	eReadMode   	: E_BACnet_CommMode;
	fCOVIncrement	: REAL;
END_STRUCT
END_TYPE

// DUTs/Types/Remote/[Internal]/ST_BACnetRM_ReqPtr
{attribute 'hide'} // [Workaround] Not hidden when lib is included

TYPE INTERNAL ST_BACnetRM_ReqPtr :
UNION
	nByte : POINTER TO BYTE;
	pPtr : PVOID;
	iReq : I_BACnetRM_BaseReq;
	
	fbBase : POINTER TO FB_BACnetRM_ReqBasic;
	fbCov : POINTER TO FB_BACnetRM_ReqCov;
	fbRead : POINTER TO FB_BACnetRM_ReqRead;
	fbRpm : POINTER TO FB_BACnetRM_ReqRpm;
	fbWrite : POINTER TO FB_BACnetRM_ReqWrite;
	fbWpm : POINTER TO FB_BACnetRM_ReqWpm;
END_UNION
END_TYPE

// DUTs/Types/Remote/[Internal]/ST_BACnetRM_RpmListEntry
{attribute 'hide'} // [Workaround] Not hidden when lib is included

{attribute 'enable_dynamic_creation'}
TYPE INTERNAL ST_BACnetRM_RpmListEntry :
STRUCT
	nEntrySize 	: DWORD;					// 0x80000000 -> next entry
	tObjectID	: T_BACnet_ObjectIdentifier;
	ePropID		: E_BACnetPropIdentifier;
	nValidBits	: DWORD;
	nArrayIndex	: DWORD;
	nPriority	: DWORD;
END_STRUCT
END_TYPE

// DUTs/Types/Remote/[Internal]/ST_BACnetRM_ScanParameter
{attribute 'hide'} // [Workaround] Not hidden when lib is included

TYPE INTERNAL ST_BACnetRM_ScanParameter :
STRUCT
	bRescrictID	 : BIT;
	bRestrictNet : BIT;
	bLocalBroadcast : BIT;
	nNetNr : UINT;
	nStartID : UDINT;
	nEndID : UDINT;
END_STRUCT
END_TYPE

// DUTs/Types/Remote/[Internal]/ST_BACnetRM_WriteEntry
{attribute 'hide'} // [Workaround] Not hidden when lib is included

{attribute 'enable_dynamic_creation'}
TYPE INTERNAL ST_BACnetRM_WriteEntry :
STRUCT
	iObject 		: I_BACnetRM_BaseObject;
	ePropID 		: E_BACnetPropIdentifier;
	
	iWriteFB 		: I_BACnetRM_BasicReq;
	
	nData 			: UDINT;
	pData 			: PVOID;
	pEnable 		: POINTER TO BOOL;
	pNull 			: POINTER TO BOOL;
	nIndex 			: UDINT := 16#FFFFFFFF;
	fCOVIncrement	: REAL := 0.0;
	nPriority 		: UDINT := 16;
END_STRUCT
END_TYPE

// DUTs/Types/Remote/ST_BACnetRM_ScanResult
TYPE ST_BACnetRM_ScanResult :
STRUCT
	tDeviceObjIdentifier	: T_BACnet_ObjectIdentifier;
	aNetAddress				: ARRAY [0..11] OF BYTE;
	nNetID					: UINT;
	{attribute 'hide'}
	nReserve1				: UINT;
	tIPAddr					: IPADDR;	
	nUDPPort				: UINT;		
	nVendorID				: UINT;
	tMaxAddr				: ETHERNET_ADDRESS;
END_STRUCT
END_TYPE

// TEST/TestPackage/Templates/HeatSupply/E_xEnergyLvl
{attribute 'qualified_only'}
TYPE E_xEnergyLvl :
(
	Protection		:= 1,
	Economy			:= 2,
	Comfort			:= 3
) UDINT;
END_TYPE

// TEST/TestPackage/Templates/HeatSupply/E_xEnergyLvlA
{attribute 'qualified_only'}
TYPE E_xEnergyLvlA :
(
	Automatic		:= 1,
	Protection		:= (E_xEnergyLvl.Protection + Automatic),
	Economy			:= (E_xEnergyLvl.Economy + Automatic),
	Comfort			:= (E_xEnergyLvl.Comfort + Automatic)
) UDINT;
END_TYPE

// GVLs/BACnet_Globals
{attribute 'qualified_only'}
VAR_GLOBAL
	{region 'Default Objects'}
		DefaultAdapter					: FB_BACnet_Adapter;									// Global linkable BACnet adapter
		DefaultServer					: FB_BACnet_Server;										// Global linkable BACnet device
	{endregion}
END_VAR
VAR_GLOBAL CONSTANT
	{region 'Commands'}
		sCmd_ConcatTitle				: STRING(5)									:= '\/';	// Command for inheriting path in entered title.
	{endregion}

	{region 'Placeholder'}
		{region 'Type Ranges'}
			nRange_ObjectTypeFirst		: INT										:= E_BACnetObjType.ObjAnalogInput;
			nRange_ObjectTypeLast		: INT										:= E_BACnetObjType.ObjChannel;
			nRange_ObjectTypeCount		: INT										:= (nRange_ObjectTypeLast - nRange_ObjectTypeFirst + 1);
		{endregion}
		{region 'Types'}
			nBACnetString_MaxLength		: INT										:= 256;
			nBACnetObjId_None			: T_BACnet_ObjectIdentifier					:= 16#FFFFFFFF;
			nBACnetInstId_Auto			: T_BACnet_ObjectIdentifier					:= 16#003FFFFF;
		{endregion}
	{endregion}

	{region 'Object specification'}
		aSpec_ObjectTypeShortcut		: ARRAY [nRange_ObjectTypeFirst .. nRange_ObjectTypeLast] OF STRING(6) := [
											(* 	AnalogInput							*)	'AI',
											(* 	AnalogOutput						*)	'AO',
											(* 	AnalogValue							*)	'AV',
											(* 	BinaryInput							*)	'BI',
											(* 	BinaryOutput						*)	'BO',
											(* 	BinaryValue							*)	'BV',
											(* 	Calendar							*)	'CAL',
											(* 	Command								*)	'CMD',
											(* 	Device								*)	'DEV',
											(* 	EventEnrollment						*)	'EE',
											(* 	File								*)	'FILE',
											(* 	Group								*)	'GROUP',
											(* 	Loop								*)	'LOOP',
											(* 	MultiStateInput						*)	'MI',
											(* 	MultiStateOutput					*)	'MO',
											(* 	NotificationClass					*)	'NC',
											(* 	Program								*)	'PROG',
											(* 	Schedule							*)	'SCHED',
											(* 	Averaging							*)	'AVG',
											(* 	MultiStateValue						*)	'MV',
											(* 	TrendLog							*)	'TLOG',
											(* 	LifeSafetyPoint						*)	'LSP',
											(* 	LifeSafetyZone						*)	'LSZ',
											(* 	Accumulator							*)	'ACC',
											(* 	PulseConverter						*)	'PC',
											(* 	EventLog							*)	'ELOG',
											(* 	GlobalGroup							*)	'GGROUP',
											(* 	TrendLogMultiple					*)	'TLM',
											(* 	LoadControl							*)	'LOAD',
											(* 	StructuredView						*)	'VIEW',
											(* 	AccessDoor							*)	'DOOR',
											(* 	<Reserved>							*)	'',
											(* 	AccessCredential					*)	'AC',
											(* 	AccessPoint							*)	'AP',
											(* 	AccessRights						*)	'AR',
											(* 	AccessUser							*)	'AU',
											(* 	AccessZone							*)	'AZ',
											(* 	CredentialDataInput					*)	'CDI',
											(* 	NetworkSecurity						*)	'NS',
											(* 	BitStringValue						*)	'BIV',
											(* 	CharacterStringValue				*)	'CV',
											(* 	DatePatternValue					*)	'DPV',
											(* 	DateValue							*)	'DV',
											(* 	DateTimePatternValue				*)	'DTPV',
											(* 	DateTimeValue						*)	'DV',
											(* 	IntegerValue						*)	'IV',
											(* 	LargeAnalogValue					*)	'LAV',
											(* 	OctetStringValue					*)	'OV',
											(* 	PositiveIntegerValue				*)	'PIV',
											(* 	TimePatternValue					*)	'TPV',
											(* 	TimeValue							*)	'TV',
											(* 	NetworkPort							*)	'NP',
											(* 	AlertEnrollment						*)	'AE',
											(* 	Channel								*)	'C'
										];
	{endregion}
	{region 'Error specification'}
		aSpec_ErrorType					: ARRAY [E_BACnet_ErrorType.First .. E_BACnet_ErrorType.Last] OF STRING := [
											(* 	eError								*)	'Error',
											(* 	eReject								*)	'Reject',
											(* 	eAbort								*)	'Abort'
										];
		aSpec_ErrorClass				: ARRAY [E_BACnet_ErrorClass.First .. E_BACnet_ErrorClass.Last] OF STRING := [
											(* 	eDevice								*)	'Device',
											(* 	eObject								*)	'Object',
											(* 	eProperty							*)	'Property',
											(* 	eResources							*)	'Resources',
											(* 	eSecurity							*)	'Security',
											(* 	eServices							*)	'Services',
											(* 	eVt									*)	'Vt',
											(* 	eCommunication						*)	'Communication'
										];
		aSpec_ErrorCode					: ARRAY [E_BACnet_ErrorCode.First .. E_BACnet_ErrorCode.Last] OF STRING := [
											(* 	eOther								*)	'Other',
											(* 	eAuthenticationFailed				*)	'Authentication failed',
											(* 	eConfigurationInProgress			*)	'Configuration in progress',
											(* 	eDeviceBusy							*)	'Device busy',
											(* 	eDynamicCreationNotSupported		*)	'Dynamic creation not supported',
											(* 	eFileAccessDenied					*)	'File access denied',
											(* 	eIncompatibleSecurityLevels			*)	'Incompatible security levels',
											(* 	eInconsistentParameters				*)	'Inconsistent parameters',
											(* 	eInconsistentSelectionCriterion		*)	'Inconsistent selection criterion',
											(* 	eInvalidDataType					*)	'Invalid data type',
											(* 	eInvalidFileAccessMethod			*)	'Invalid file access method',
											(* 	eInvalidFileStartPosition			*)	'Invalid file start position',
											(* 	eInvalidOperatorName				*)	'Invalid operator name',
											(* 	eInvalidParameterDataType			*)	'Invalid parameter data type',
											(* 	eInvalidTimeStamp					*)	'Invalid time stamp',
											(* 	eKeyGenerationError					*)	'Key generation error',
											(* 	eMissingRequiredParameter			*)	'Missing required parameter',
											(* 	eNoObjectsOfSpecifiedType			*)	'No objects of specified type',
											(* 	eNoSpaceForObject					*)	'No space for object',
											(* 	eNoSpaceToAddListElement			*)	'No space to add list element',
											(* 	eNoSpaceToWriteProperty				*)	'No space to write property',
											(* 	eNoVTSessionsAvailable				*)	'No vt sessions available',
											(* 	ePropertyIsNotAList					*)	'Property is not a list',
											(* 	eObjectDeletionNotPermitted			*)	'Object deletion not permitted',
											(* 	eObjectIdentifierAlreadyExists		*)	'ObjectIdentifier already exists',
											(* 	eOperationalProblem					*)	'Operational problem',
											(* 	ePasswordFailure					*)	'Password failure',
											(* 	eReadAccessDenied					*)	'Read access denied',
											(* 	eSecurityNotSupported				*)	'Security not supported',
											(* 	eServiceRequestDenied				*)	'Service request denied',
											(* 	eTimeout							*)	'Timeout',
											(* 	eUnknownObject						*)	'Unknown object',
											(* 	eUnknownProperty					*)	'Unknown property',
											(* 	<Reserve>							*)	'',
											(* 	eUnknownVTClass						*)	'Unknown vt class',
											(* 	eUnknownVTSession					*)	'Unknown vt session',
											(* 	eUnsupportedObjectType				*)	'Unsupported object type',
											(* 	eValueOutOfRange					*)	'Value out of range',
											(* 	eVtSessionAlreadyClosed				*)	'Vt session already closed',
											(* 	eVtSessionTerminationFailure		*)	'Vt session termination failure',
											(* 	eWriteAccessDenied					*)	'Write access denied',
											(* 	eCharacterSetNotSupported			*)	'Character set not supported',
											(* 	eInvalidArrayIndex					*)	'Invalid array index',
											(* 	eCovSubscriptionFailed				*)	'COV subscription failed',
											(* 	eNotCovProperty						*)	'Not COV property',
											(* 	eOptionalFunctionalityNotSupported	*)	'Optional functionality not supported',
											(* 	eInvalidConfigurationData			*)	'Invalid configuration data',
											(* 	eDatatypeNotSupported				*)	'Datatype not supported',
											(* 	eDuplicateName						*)	'Duplicate name',
											(* 	eDuplicateObjectId					*)	'Duplicate object ID',
											(* 	ePropertyIsNotAnArray				*)	'Property is not an array',
											(* 	eAbortBufferOverflow				*)	'Abort buffer overflow',
											(* 	eAbortInvalidAPDUInThisState		*)	'Abort invalid apdu in this state',
											(* 	eAbortPreemptedByHigherPriorityTask	*)	'Abort preempted by higher priority task',
											(* 	eAbortSegmentationNotSupported		*)	'Abort segmentation not supported',
											(* 	eAbortProprietary					*)	'Abort proprietary',
											(* 	eAbortOther							*)	'Abort other',
											(* 	eInvalidTag							*)	'Invalid tag',
											(* 	eNetworkDown						*)	'Network down',
											(* 	eRejectBufferOverflow				*)	'Reject buffer overflow',
											(* 	eRejectInconsistentParameters		*)	'Reject inconsistent parameters',
											(* 	eRejectInvalidParameterDataType		*)	'Reject invalid parameter data type',
											(* 	eRejectInvalidTag					*)	'Reject invalid tag',
											(* 	eRejectMissingRequiredParameter		*)	'Reject missing required parameter',
											(* 	eRejectParameterOutOfRange			*)	'Reject parameter out of range',
											(* 	eRejectTooManyArguments				*)	'Reject too many arguments',
											(* 	eRejectUndefinedEnumeration			*)	'Reject undefined enumeration',
											(* 	eRejectUnrecognizedService			*)	'Reject unrecognized service',
											(* 	eRejectProprietary					*)	'Reject proprietary',
											(* 	eRejectOther						*)	'Reject other',
											(* 	eUnknownDevice						*)	'Unknown device',
											(* 	eUnknownRoute						*)	'Unknown route',
											(* 	eValueNotInitialized				*)	'Value not initialized',
											(* 	eInvalidEventState					*)	'Invalid event state',
											(* 	eNoAlarmConfigured					*)	'No alarm configured',
											(* 	eLogBufferFull						*)	'Log buffer full',
											(* 	eLoggedValuePurged					*)	'Logged value purged',
											(* 	eNoPropertySpecified				*)	'No property specified',
											(* 	eNotConfiguredForTriggeredLogging	*)	'Not configured for triggered logging',
											(* 	eUnknownSubscription				*)	'Unknown subscription',
											(* 	eParameterOutOfRange				*)	'Parameter out of range',
											(* 	eListElementNotFound				*)	'List element not found',
											(* 	eBusy								*)	'Busy',
											(* 	eCommunicationDisabled				*)	'Communication disabled',
											(* 	<Reserve>							*)	38(''),
											(* 	eUnknownFileSize					*)	'Unknown file size',
											(* 	eAbortAPDUTooLong					*)	'Abort Apdu Too Long',
											(* 	eAbortApplicationExceededReplyTime	*)	'Abort Application Exceeded Reply Time',
											(* 	eAbortOutOfResources				*)	'Abort Out Of Resources',
											(* 	eAbortTsmTimeout					*)	'Abort Tsm Timeout',
											(* 	eAbortWindowSizeOutOfRange			*)	'Abort Window Size Out Of Range',
											(* 	eFileFull							*)	'File Full',
											(* 	eInconsistentConfiguration			*)	'Inconsistent Configuration',
											(* 	eInconsistentObjectType				*)	'Inconsistent object type',
											(* 	eInternalError						*)	'Internal Error',
											(* 	eNotConfigured						*)	'Not Configured',
											(* 	eOutOfMemory						*)	'Out Of Memory'
										];
		aSpec_RejectReason				: ARRAY [E_BACnet_RejectReason.First .. E_BACnet_RejectReason.Last] OF STRING := [
											(* 	eOther								*)	'Other',
											(* 	eBufferOverflow						*)	'Buffer overflow',
											(* 	eInconsistentParameters				*)	'Inconsistent parameters',
											(* 	eInvalidParameterDataType			*)	'Invalid parameter data type',
											(* 	eInvalidTag							*)	'Invalid tag',
											(* 	eMissingRequiredParameter			*)	'Missing required parameter',
											(* 	eParameterOutOfRange				*)	'Parameter out of range',
											(* 	eTooManyArguments					*)	'Too many arguments',
											(* 	eUndefinedEnumeration				*)	'Undefined enumeration',
											(* 	eUnrecognizedService				*)	'Unrecognized service'
										];
		aSpec_AbortReason				: ARRAY [E_BACnet_AbortReason.First .. E_BACnet_AbortReason.Last] OF STRING := [
											(* 	eOther								*)	'Other',
											(* 	eBufferOverflow						*)	'Buffer overflow',
											(* 	eInvalidAPDUInThisState				*)	'Invalid apdu in this state',
											(* 	ePreemptedByHigherPriorityTask		*)	'Preempted by higher priority task',
											(* 	eSegmentationNotSupported			*)	'Segmentation not supported',
											(* 	<Reserve>							*)	2(''),
											(* 	eWindowSizeOutOfRange				*)	'Window size out of range',
											(* 	eApplicationExceededReplyTime		*)	'Application exceeded reply time',
											(* 	eOutOfResources						*)	'Out of resources',
											(* 	eTSMTimeout							*)	'Tsm timeout',
											(* 	eAPDUTooLong						*)	'Apdu too long'
										];
	{endregion}
END_VAR
VAR_GLOBAL CONSTANT INTERNAL
	{region 'Placeholder'}
		{region 'AMS'}
			tInvalidAmsNetId			: T_AmsNetId						:= '0.0.0.0.0.0';
		{endregion}
		{region 'Types'}
			// (BETA) ... will be removed when ADS communication is removed
			{attribute 'hide'}
			nDataField_MaxExSchEntries			: UINT						:= 9;
			{attribute 'hide'}
			nDataField_MaxTimeValues			: UINT						:= 9;
			{attribute 'hide'}
			nDataField_MaxObjIdList				: UINT						:= 1999;
			{attribute 'hide'}
			nDataField_MaxLogBufferEntries		: UINT						:= 499;
			{attribute 'hide'}
			nDataField_MaxEventLogBufferEntries	: UINT						:= 500;
		{endregion}
	{endregion}
END_VAR

VAR_GLOBAL
	{region 'Internal'}
		// 8kByte common ADS buffer used by function blocks that access BACnet over ADS
		// [IMPORTANT] Use type "UDINT" instead of "BYTE" to ensure correct alignment!
		{attribute 'hide'}
		aDefaultBuffer					: ARRAY [0 .. (BACnet_Param.nADS_BufferSize/4)] OF UDINT;
	{endregion}
END_VAR

// GVLs/BACnet_Param
{attribute 'qualified_only'}
VAR_GLOBAL CONSTANT
	{region 'ADS'}
		tADS_TimeOut							: TIME						:= T#15S;
		nADS_BufferSize							: INT						:= 25535;								// Default 24 kByte buffer
	{endregion}
	{region 'Priorities'}
		ePrio_LifeSafety 						: E_BACnet_Priority			:= E_BACnet_Priority.eP1;
		ePrio_Critical							: E_BACnet_Priority			:= E_BACnet_Priority.eP5;
		ePrio_ManLocal							: E_BACnet_Priority			:= E_BACnet_Priority.eP7;
		ePrio_ManOperator 						: E_BACnet_Priority			:= E_BACnet_Priority.eP8;
		ePrio_Program 	 						: E_BACnet_Priority			:= E_BACnet_Priority.eP15;
		ePrio_Default	 	 					: E_BACnet_Priority			:= E_BACnet_Priority.eDefault;			// No priority used

		eRemotePrio_Default						: E_BACnet_Priority			:= E_BACnet_Priority.eP8;				// Default priority for priority enabled remote-objects
	{endregion}
		
	{region 'Event-Management'}
		sEvtMgmt_AckMsgRemote					: STRING					:= 'Acknowledged by remote user.';		// Text to indicate acknowledgement via remote access.
		sEvtMgmt_AckMsgPLC						: STRING					:= 'Acknowledged by PLC.';				// Text to indicate acknowledgement via PLC logic.
	{endregion}
	{region 'Titles'}
		sSeparator_ObjectName					: STRING					:= '_';									// Separator to be used when building Inherited object names
		sSeparator_Description					: STRING					:= ' - ';								// Separator to be used when building Inherited descriptions
		sSeparator_EventMessageText				: STRING					:= ' - ';								// Separator to be used when building Inherited event message texts
	{endregion}
		 
	{region 'Objects'}
		{region 'General'}
			nStateText_Length					: UDINT						:= 40;									// Max. count of string characters in state texts (e.g. Multustate-StateText, Binary-In/ActiveText)
			bStateText_WriteProtect				: BOOL						:= FALSE;
		{endregion}
		{region 'Multistate'}
			nMultistate_StateCount				: UDINT						:= 12;									// Count of state entries
			{attribute 'TcEncoding':='UTF-8'}
			sMultistate_DefaultStateText		: T_BACnet_StateTextArray	:= [ 'State 1', 'State 2', 'State 3' ];
		{endregion}
		{region 'Log'}  
			nLog_BufferEntryCount				: UDINT						:= 500;
					  
			nTLM_ReferenceCount					: UDINT						:= 8;
		{endregion}
		{region 'Loop'}
			nLoop_PrioForWriting				: UDINT						:= 16;
		{endregion}
		{region 'Calendar'}
			nCal_DateListCount					: INT						:= 24;									// Count of date list entries ('T_BACnet_CalendarDateList')
		{endregion}
		{region 'NC'}
			nNC_RecipientListSize				: INT						:= 8;									// Count of recipient entries
		{endregion}
		{region 'Scheduler'}
			nSched_PrioForWriting				: UDINT						:= 16;
						  
			nSched_EntryCount					: INT						:= 6;									// Count of entries in a weekday ('T_BACnet_SchedWeek') or an exception ('ST_BACnet_SchedCalendar' / 'ST_BACnet_SchedException')
			nSched_CalendarCount				: INT						:= 3;									// Count of calendar references ('T_BACnet_SchedCalendar')
			nSched_ExceptionCount				: INT						:= 24;									// Count of exceptions ('T_BACnet_SchedException')

			nSched_ReferenceCount				: UDINT						:= 2;
					  
			eSched_BType						: E_BACnet_SchedBType		:= E_BACnet_SchedBType.eBinaryPV;		// Internal datatype of boolean schedulers
		{endregion}
		{region 'Event Enrollment'}
			nEE_EventParameter_BinaryCodedSize	: UDINT						:= 100;
		{endregion}
	{endregion}
END_VAR

// TEST/TestPackage/Templates/Const
{attribute 'qualified_only'}
VAR_GLOBAL CONSTANT
	rClsZero        : REAL := 0.00001;//Comparison value to prevent a division by zero
						
	nNoActvPrio	: UDINT	:= 4294967295;//Value of the constant indicates that no priority is active	
	
	nTiSec        : UDINT := 4294966;
	nTiMin        : UDINT := 71582;

	wSUNDAY         : WORD := 0;//Constant value for Sunday
	wMONDAY         : WORD := 1;//Constant value for Monday
	wTUESDAY        : WORD := 2;//Constant value for Tuesday
	wWEDNESDAY      : WORD := 3;//Constant value for Wednesday
	wTHURSDAY       : WORD := 4;//Constant value for Thursday
	wFRIDAY         : WORD := 5;//Constant value for Friday
	wSATURDAY       : WORD := 6;//Constant value for Saturday

	TimeValue24h_ms : UDINT := 86400000;//Time value for 24 hours in ms
END_VAR

// Version/Global_Version
{attribute 'TcGenerated'}
{attribute 'no-analysis'}
{attribute 'linkalways'}
// This function has been automatically generated from the project information.
VAR_GLOBAL CONSTANT
	{attribute 'const_non_replaced'}
	stLibVersion_Tc3_BACnetRev14 : ST_LibVersion := (iMajor := 4, iMinor := 0, iBuild := 18, iRevision := 1, nFlags := 0, sVersion := '4.0.18.1');
END_VAR

// DUTs/Interfaces/Remote/Objects/[Base]/I_BACnetRM_Object
INTERFACE I_BACnetRM_Object EXTENDS I_BACnetRM_BaseObject

END_INTERFACE

// DUTs/Interfaces/Remote/Objects/[Internal]/I_BACnetRM_BaseObject
INTERFACE I_BACnetRM_BaseObject EXTENDS __SYSTEM.IQueryInterface

{attribute 'hide'}
METHOD OnCOV
VAR_INPUT
	ePropID		: E_BACnetPropIdentifier;
END_VAR
END_METHOD

{attribute 'hide'}
METHOD OnReqError
VAR_INPUT
	iRequest		: I_BACnetRM_BaseReq;
	stResult		: POINTER TO SendDataRequestResult;
	sLogCode		: STRING			:= '';
END_VAR
END_METHOD

PROPERTY Error : BOOL
GET
END_GET
END_PROPERTY

PROPERTY ObjectID : T_BACnet_ObjectIdentifier
GET
END_GET
END_PROPERTY

PROPERTY ObjectInstance : UDINT
GET
END_GET
END_PROPERTY

PROPERTY ObjectType : E_BACnetObjType
GET
END_GET
END_PROPERTY

PROPERTY ReadMode : E_BACnet_CommMode
GET
END_GET
SET
END_SET
END_PROPERTY

END_INTERFACE

// DUTs/Interfaces/Remote/Requests/[Base]/I_BACnetRM_BaseReq
{attribute 'c++_compatible'}
INTERFACE I_BACnetRM_BaseReq

{attribute 'hide'}
METHOD Send : BOOL
VAR_INPUT
END_VAR
END_METHOD

METHOD GetRequestType : E_BACnetRM_RequestType
VAR_INPUT
END_VAR
END_METHOD

METHOD IsReady : BOOL
VAR_INPUT
END_VAR
END_METHOD

END_INTERFACE

// DUTs/Interfaces/Remote/Objects/[Internal]/I_BACnetRM_ObjectOwner
{attribute 'hide'}
INTERFACE I_BACnetRM_ObjectOwner EXTENDS __SYSTEM.IQueryInterface

{attribute 'hide'}
METHOD OnBACnetRMObjectCOV
VAR_INPUT
	ePropID		: E_BACnetPropIdentifier;
END_VAR
END_METHOD

{attribute 'hide'}
METHOD OnBACnetRMObjectStateChanged
END_METHOD

{attribute 'suppress_wrn_C0410'}
{attribute 'hide'}
PROPERTY LogMsg : REFERENCE TO FB_BA_LogMessage
GET
END_GET
END_PROPERTY

END_INTERFACE

// DUTs/Interfaces/Remote/Requests/[Base]/I_BACnetRM_BasicReq
INTERFACE I_BACnetRM_BasicReq EXTENDS __SYSTEM.IQueryInterface

{attribute 'hide'}
METHOD SetError
END_METHOD

{attribute 'hide'}
METHOD SetReady
END_METHOD

END_INTERFACE

// DUTs/Interfaces/Server/[Base]/I_BACnet_Object
INTERFACE I_BACnet_Object EXTENDS I_BACnet_BaseObject

{attribute 'hide'}
PROPERTY NextSibling : I_BACnet_Object
GET
END_GET
SET
END_SET
END_PROPERTY

{attribute 'hide'}
PROPERTY PrevSibling : I_BACnet_Object
GET
END_GET
SET
END_SET
END_PROPERTY

PROPERTY IsDynamic : BOOL
GET
END_GET
END_PROPERTY

PROPERTY Parent : I_BACnet_View
GET
END_GET
SET
END_SET
END_PROPERTY

PROPERTY Description : T_MaxString
GET
END_GET
SET
END_SET
END_PROPERTY

PROPERTY ObjectName : T_MaxString
GET
END_GET
SET
END_SET
END_PROPERTY

END_INTERFACE

// DUTs/Interfaces/Server/[Internal]/I_BACnet_BaseObject
{attribute 'hide'}
INTERFACE I_BACnet_BaseObject EXTENDS I_BA_SupplementObject

{attribute 'hide'}
PROPERTY NextObject : I_BACnet_BaseObject
GET
END_GET
SET
END_SET
END_PROPERTY

PROPERTY Error : BOOL
GET
END_GET
END_PROPERTY

PROPERTY ObjectID : T_BACnet_ObjectIdentifier
GET
END_GET
END_PROPERTY

PROPERTY ObjectInstance : UDINT
GET
END_GET
END_PROPERTY

PROPERTY ObjectType : E_BACnetObjType
GET
END_GET
END_PROPERTY

PROPERTY Ready : BOOL
GET
END_GET
END_PROPERTY

METHOD ReadProperty : HRESULT
VAR_INPUT
	ePropID : E_BACnetPropIdentifier;
	pData : PVOID;
	nData : POINTER TO DINT;
END_VAR
END_METHOD

METHOD SyncPropertyCOV : BOOL
VAR_INPUT
	ePropertyID : E_BACnetPropIdentifier;
	bCOVTrig : POINTER TO BOOL;
END_VAR
END_METHOD

METHOD WriteProperty : HRESULT
VAR_INPUT
	ePropID : E_BACnetPropIdentifier;
	pData : PVOID;
	nData : DINT;
END_VAR
END_METHOD

END_INTERFACE

// DUTs/Interfaces/Server/Misc/I_BACnet_View
INTERFACE I_BACnet_View EXTENDS I_BACnet_Object

{attribute 'hide'}
METHOD AddObject : BOOL
VAR_INPUT
	iObject			: I_BACnet_Object;
END_VAR
VAR_OUTPUT
	nResultIndex	: DINT;
END_VAR
END_METHOD

{attribute 'hide'}
METHOD RemoveObject : BOOL
VAR_INPUT
	iObject			: I_BACnet_Object;
END_VAR
END_METHOD

METHOD FindObject : BOOL
VAR_INPUT
	iObject			: I_BACnet_Object;
END_VAR
VAR_IN_OUT
	nResultIndex	: DINT;
END_VAR
END_METHOD

END_INTERFACE

// DUTs/Interfaces/Server/[Internal]/I_BACnet_ObjectOwner
{attribute 'hide'}
INTERFACE I_BACnet_ObjectOwner EXTENDS __SYSTEM.IQueryInterface

{attribute 'suppress_wrn_C0410'}
{attribute 'hide'}
PROPERTY LogMsg : REFERENCE TO FB_BA_LogMessage
GET
END_GET
END_PROPERTY

{attribute 'hide'}
PROPERTY SymbolName : POINTER TO STRING
GET
END_GET
END_PROPERTY

{attribute 'hide'}
PROPERTY SymbolPath : POINTER TO T_MaxString
GET
END_GET
END_PROPERTY

{attribute 'hide'}
METHOD OnBACnetObjectStateChanged
VAR_INPUT
	tState			: TCOM_STATE;
END_VAR
END_METHOD

END_INTERFACE

// DUTs/Interfaces/Server/Misc/I_BACnet_Cal
INTERFACE I_BACnet_Cal EXTENDS I_BACnet_Object

END_INTERFACE

// POUs/Dynamic Objects/FB_BACnet_DynObjectManager
// Management of dynamically object generation.
// [Abilities]
// - Creating standard and derived objects dynamically.
// - Deleting previously created objects.
// - Automatically deletes created objects when system shuts down.
// - Automatically call created objects (Optional)
FUNCTION_BLOCK FB_BACnet_DynObjectManager
VAR_INPUT CONSTANT
	{region 'Variable Parameters'}
		{attribute 'parameterCategory':='General'}
		bCycleObjects : BOOL;								// [Optional] Call dynamically created objects cyclic (if no other calling-implementation is intended)
	{endregion}
END_VAR
VAR
	{region 'Linked Object-List'
		{attribute 'hide'}
		iFirstChild			: I_BACnet_Object;
		{attribute 'hide'}
		iLastChild			: I_BACnet_Object;
		bCreatedObjects		: UDINT;
	{endregion}
	{region 'Internal'}
		{attribute 'hide'}
		{attribute 'no_copy'}
		Server				: REFERENCE TO FB_BACnet_Server := BACnet_Globals.DefaultServer;
		{attribute 'hide'}
		nUpdateCount 		: UDINT := 0;
	{endregion}
END_VAR
VAR_STAT
	{region 'Temporary'}
		{attribute 'hide'}
		_iObj				: I_BACnet_Object;
	{endregion}	
END_VAR

// Update device:
IF (Server.nUpdateCount = nUpdateCount) THEN
	Server();
END_IF
nUpdateCount := Server.nUpdateCount;

IF (TwinCAT_SystemInfoVarList._AppInfo.ShutdownInProgress) THEN
	Reset();
ELSE
	IF (bCycleObjects) THEN
		EvaluateStructure(E_BACnet_EvaluationMode.eCycle, 0, TRUE);
	END_IF
END_IF

METHOD PRIVATE EvaluateStructure
VAR_INPUT
	eMode			: E_BACnet_EvaluationMode;
	iObject			: I_BACnet_Object			:= 0;
	bRecursive		: BOOL						:= FALSE;
END_VAR
VAR
	_iObj			: I_BACnet_Object;
	_iTemp			: I_BACnet_Object;
	_fbView			: POINTER TO FB_BACnet_View;
END_VAR
VAR_STAT
	{region 'Temporary'}
		{attribute 'hide'}
		_fbObject	: POINTER TO FB_BACnet_Object;
	{endregion}	
END_VAR
IF (iObject = 0) THEN
	// Iterate though root objects:
	_iObj := iFirstChild;
	WHILE (_iObj <> 0) DO
		_iTemp := _iObj.NextSibling;
		THIS^.EvaluateStructure(eMode, _iObj, bRecursive);
		_iObj := _iTemp;
	END_WHILE;
ELSE
	// Pre-Evaluation treatment:
	CASE (eMode) OF
		E_BACnet_EvaluationMode.eCycle:
			iObject.OnCycle(FALSE);
	END_CASE
	
	IF (bRecursive) AND_THEN (iObject.ObjectType = E_BACnetObjType.ObjStructuredView) AND_THEN (__QUERYPOINTER(iObject, _fbView)) THEN
		// Iterate though child-objects of 'iObject':
		_iObj := _fbView^.iFirstChild;
		WHILE (_iObj <> 0) DO
			_iTemp := _iObj.NextSibling;
			THIS^.EvaluateStructure(eMode, _iObj, bRecursive);
			_iObj := _iTemp;
		END_WHILE;
	END_IF
	
	// Post-Evaluation treatment:
	CASE (eMode) OF
		E_BACnet_EvaluationMode.eDeleteObjects:
			IF (__QUERYPOINTER(iObject, _fbObject)) THEN
				DeleteObjectEx(_fbObject);
			END_IF
	END_CASE
END_IF
END_METHOD

METHOD PRIVATE DeleteObjectEx
VAR_INPUT
	fbObject			: POINTER TO FB_BACnet_Object;
END_VAR
VAR
	_iSrv				: POINTER TO ITcIoBACnetPlcServer;
	_iObj				: POINTER TO ITcIoBACnetPlcObject;
END_VAR
_iSrv := ADR(fbObject^.ipSrv);
_iObj := ADR(fbObject^.ipObj);

IF (_iSrv^.DeletePlcObjectRT(_iObj) <> S_OK) THEN
	F_BA_LogMessage1(ADSLOG_MSGTYPE_WARN, 'DO46', 'Dynamic PLC object deleted, but failed to delete object "%s" from stack!', F_STRING(fbObject^.sObjectName));
END_IF

__DELETE(fbObject);
bCreatedObjects := (bCreatedObjects-1);
END_METHOD

// Called after online change.
{attribute 'call_after_online_change_slot' := '10'}
METHOD PROTECTED OnPostOnlineChange
Reset();
END_METHOD

// Create an object dynamically.
METHOD CreateObject : BOOL
VAR_IN_OUT
	fbResult			: POINTER TO FB_BACnet_Object;
END_VAR
VAR_INPUT
	eObjectType			: E_BACnet_CreateObjType;
	nObjectInstance		: UDINT							:= BACnet_Globals.nBACnetInstId_Auto;
	sObjectName			: T_MaxString;
	sDescription		: T_MaxString;
	fbParent			: POINTER TO FB_BACnet_View		:= 0;
END_VAR
VAR
	_uObj				: U_BACnet_CreateObj;
END_VAR
// Evaluate type:
CASE (eObjectType) OF
	E_BACnet_CreateObjType.eAnalogInputRaw:			_uObj.AIRaw := __NEW(FB_BACnet_AI_Raw);
	E_BACnet_CreateObjType.eAnalogOutputRaw:		_uObj.AORaw := __NEW(FB_BACnet_AO_Raw);
	E_BACnet_CreateObjType.eAnalogOutputRaw5P:		_uObj.AORaw5P := __NEW(FB_BACnet_AO_Raw5P);
	E_BACnet_CreateObjType.eAnalogValue:			_uObj.AV := __NEW(FB_BACnet_AV);
	E_BACnet_CreateObjType.eAnalogValue5P:			_uObj.AV5P := __NEW(FB_BACnet_AV_5P);
	E_BACnet_CreateObjType.eAnalogValueDisp:		_uObj.AVDisp := __NEW(FB_BACnet_AV_Disp);
	E_BACnet_CreateObjType.eAnalogValueSetp:		_uObj.AVSetp := __NEW(FB_BACnet_AV_Setp);
	
	E_BACnet_CreateObjType.eBinaryInputRaw:			_uObj.BIRaw := __NEW(FB_BACnet_BI_Raw);
	E_BACnet_CreateObjType.eBinaryOutputRaw:		_uObj.BORaw := __NEW(FB_BACnet_BO_Raw);
	E_BACnet_CreateObjType.eBinaryOutputRaw5P:		_uObj.BORaw5P := __NEW(FB_BACnet_BO_Raw5P);
	E_BACnet_CreateObjType.eBinaryValue:			_uObj.BV := __NEW(FB_BACnet_BV);
	E_BACnet_CreateObjType.eBinaryValue5P:			_uObj.BV5P := __NEW(FB_BACnet_BV_5P);
	E_BACnet_CreateObjType.eBinaryValueDisp:		_uObj.BVDisp := __NEW(FB_BACnet_BV_Disp);
	E_BACnet_CreateObjType.eBinaryValueSetp:		_uObj.BVSetp := __NEW(FB_BACnet_BV_Setp);
	
	E_BACnet_CreateObjType.eMultistateInputRaw:		_uObj.MIRaw := __NEW(FB_BACnet_MI_Raw);
	E_BACnet_CreateObjType.eMultistateOutputRaw:	_uObj.MORaw := __NEW(FB_BACnet_MO_Raw);
	E_BACnet_CreateObjType.eMultistateOutputRaw5P:	_uObj.MORaw5P := __NEW(FB_BACnet_MO_Raw5P);
	E_BACnet_CreateObjType.eMultistateValue:		_uObj.MV := __NEW(FB_BACnet_MV);
	E_BACnet_CreateObjType.eMultistateValue5P:		_uObj.MV5P := __NEW(FB_BACnet_MV_5P);
	E_BACnet_CreateObjType.eMultistateValueDisp:	_uObj.MVDisp := __NEW(FB_BACnet_MV_Disp);
	E_BACnet_CreateObjType.eMultistateValueSetp:	_uObj.MVSetp := __NEW(FB_BACnet_MV_Setp);
	
	E_BACnet_CreateObjType.eCalendar:				_uObj.Clnd := __NEW(FB_BACnet_Cal);
	E_BACnet_CreateObjType.eDevice:					_uObj.Device := __NEW(FB_BACnet_Device);
	E_BACnet_CreateObjType.eFile:					_uObj.File := __NEW(FB_BACnet_File);
	E_BACnet_CreateObjType.eLoop:					_uObj.Loop := __NEW(FB_BACnet_Loop);
	E_BACnet_CreateObjType.eNotificationClass:		_uObj.NC := __NEW(FB_BACnet_NC);
	E_BACnet_CreateObjType.eProg:					_uObj.Prog := __NEW(FB_BACnet_Prog);
	E_BACnet_CreateObjType.eScheduleAnalog:			_uObj.SchedA := __NEW(FB_BACnet_SchedA);
	E_BACnet_CreateObjType.eScheduleBinary:			_uObj.SchedB := __NEW(FB_BACnet_SchedB);
	E_BACnet_CreateObjType.eScheduleMultistate:		_uObj.SchedM := __NEW(FB_BACnet_SchedM);
	E_BACnet_CreateObjType.eAccumulator:			_uObj.Acc := __NEW(FB_BACnet_Acc);
	E_BACnet_CreateObjType.ePulseConverter:			_uObj.PC := __NEW(FB_BACnet_PC);
	E_BACnet_CreateObjType.eStructuredView:			_uObj.View := __NEW(FB_BACnet_View);

ELSE
	F_BA_LogMessage1(ADSLOG_MSGTYPE_ERROR, 'CO20', 'Unsupported object type "%d"!', F_INT(eObjectType));
	RETURN;
END_CASE

IF (_uObj.Obj = 0) THEN
	F_BA_LogMessage1(ADSLOG_MSGTYPE_ERROR, 'CO25', 'Unknown error on creating dynamic object of type "%d"!', F_INT(eObjectType));
ELSE
	IF (CreateObjectEx(_uObj.Obj, nObjectInstance, sObjectName, sDescription, fbParent)) THEN
		fbResult := _uObj.Obj;
		CreateObject := TRUE;
	ELSE
		__DELETE (_uObj.Obj);
		fbResult := 0;
	END_IF
END_IF
END_METHOD

// Create an object dynamically.
// > 'fbResult' is an object, that was previously created with '__NEW()'.
//   Useful if 'fbResult' is a derived object type.
METHOD CreateObjectEx : BOOL
VAR_INPUT
	fbObject			: POINTER TO FB_BACnet_Object;
	nObjectInstance		: UDINT							:= BACnet_Globals.nBACnetInstId_Auto;
	sObjectName			: T_MaxString;
	sDescription		: T_MaxString;
	fbParent			: POINTER TO FB_BACnet_View		:= 0;
END_VAR
IF (Ready) THEN
	IF (fbObject = 0) THEN
		F_BA_LogMessage(ADSLOG_MSGTYPE_ERROR, 'CO02', 'Invalid object!');
	ELSIF (sObjectName = '') THEN
		F_BA_LogMessage1(ADSLOG_MSGTYPE_ERROR, 'CO04', 'Unable to create object due to invalid name "%s"!', F_STRINGEx(sObjectName));
	ELSIF (sDescription = '') THEN
		F_BA_LogMessage1(ADSLOG_MSGTYPE_ERROR, 'CO06', 'Unable to create object due to invalid description "%s"!', F_STRINGEx(sDescription));
	ELSIF (fbParent <> 0) AND_THEN (NOT fbParent^.IsDynamic) THEN
		F_BA_LogMessage1(ADSLOG_MSGTYPE_ERROR, 'CO08', 'Refused to create object of non-dynamic parent "%s"!', F_STRING(fbParent^.SymbolPath^));
	ELSE
		IF (fbObject^.DynamicInit(THIS, nObjectInstance, sObjectName, sDescription, fbParent)) THEN
			IF (fbParent = 0) THEN
				// Append linked object list:
				IF (iFirstChild = 0) THEN
					iFirstChild := fbObject^;
				ELSE
					iLastChild.NextSibling := fbObject^;
				END_IF
				iLastChild := fbObject^;
			END_IF
		
			bCreatedObjects := (bCreatedObjects+1);
			CreateObjectEx := TRUE;
		END_IF
	END_IF
END_IF
END_METHOD

// Delete a dynamically created object.
// > IMPORTANT: Pointers to deleted objects are invalid!
METHOD DeleteObject : BOOL
VAR_IN_OUT
	fbObject			: POINTER TO FB_BACnet_Object;
END_VAR
VAR
	_fbView				: POINTER TO FB_BACnet_View;
	_fbObject			: POINTER TO FB_BACnet_Object;
	_iObject			: I_BACnet_Object;
END_VAR
IF (fbObject = 0) THEN
	F_BA_LogMessage(ADSLOG_MSGTYPE_ERROR, 'DO02', 'Invalid dynamic object!');
ELSIF (NOT fbObject^.IsDynamic) THEN
	F_BA_LogMessage1(ADSLOG_MSGTYPE_ERROR, 'DO04', 'Refused to delete non-dynamic object "%s"!', F_STRING(fbObject^.SymbolPath^));
ELSIF (fbObject^.fbDynProducer <> THIS) THEN
	F_BA_LogMessage1(ADSLOG_MSGTYPE_ERROR, 'DO06', 'Refused to delete dynamic object "%s" that is not created by current object manager!', F_STRING(fbObject^.SymbolPath^));
ELSE
	IF (fbObject^.ObjectType = E_BACnetObjType.ObjStructuredView) THEN
		_fbView := fbObject;
		IF (_fbView^.iFirstChild <> 0) THEN
			F_BA_LogMessage1(ADSLOG_MSGTYPE_ERROR, 'DO11', 'Unable to delete dynamic object "%s" because it has existing child objects!', F_STRING(fbObject^.SymbolPath^));
			RETURN;
		END_IF
	END_IF
	
	_fbObject := fbObject;
	_iObject := _fbObject^;
	
	IF (_fbObject^.iParent = 0) THEN
		// Remove object from linked object list of current instance:
		fbObject^.RemoveFromLinkedObjList(iFirstChild, iLastChild);
	ELSE
		// Remove object from parent:
		_fbObject^.iParent.RemoveObject(_iObject);
	END_IF
	
	DeleteObjectEx(_fbObject);
	fbObject := 0;
	
	DeleteObject := TRUE;
END_IF
END_METHOD

PROPERTY Ready : BOOL
GET
Ready := Server.Operational;
END_GET
END_PROPERTY

// Delete all dynamically created objects.
METHOD Reset
// Delete all created objects:
EvaluateStructure(E_BACnet_EvaluationMode.eDeleteObjects, 0, TRUE);

iFirstChild := 0;
iLastChild := 0;
bCreatedObjects := 0;
END_METHOD

PROPERTY CreatedObjects : UDINT
GET
CreatedObjects := bCreatedObjects;
END_GET
END_PROPERTY

METHOD FB_exit : BOOL
VAR_INPUT
	bInCopyCode : BOOL; // if TRUE, the exit method is called for exiting an instance that is copied afterwards (online change).
END_VAR
Reset();
END_METHOD

END_FUNCTION_BLOCK

// POUs/Local/FB_BACnet_Server
{attribute 'no_assign'}
FUNCTION_BLOCK FB_BACnet_Server
VAR_INPUT
	bWritePersistent		: BOOL;
END_VAR
VAR_INPUT CONSTANT
	{region 'Fixed Parameters'}
		{attribute 'parameterCategory':='General'}
		Adapter	: REFERENCE TO FB_BACnet_Adapter := BACnet_Globals.DefaultAdapter;
	{endregion}
END_VAR
VAR_INPUT CONSTANT PERSISTENT
	{region 'Variable Parameters'}
		{attribute 'parameterCategory':='General'}
		bSupportBackup : BOOL;							// Support backup of PLC persistent data when BACnet backup service is used
		{attribute 'parameterCategory':='General'}
		bDisableWOC : BOOL;								// Deactivate write-on-change mechanism
		{attribute 'parameterCategory':='General'}
		tAmsPort : T_AmsPort := 1000;					// Default port when port can not be determined automatically
	{endregion}
END_VAR
VAR_INPUT CONSTANT
	{region 'Operational Parameters'}
		{attribute 'parameterCategory':='General'}
		bReset : BOOL;									// Manual trigger to reset errors
		{attribute 'parameterCategory':='General'}
		tWritePersistent : TIME := T#30M;				// Cyclic write persistent data
	{endregion}
END_VAR
VAR_OUTPUT
	nRev					: DINT := -1;				// Protocol revision no.
	stAdsConn				: ST_BACnet_AdsConnection;
	eSysStatus				: E_BACnet_DeviceStatus;
	eState					: E_BACnet_ServerState	:= E_BACnet_ServerState.eInitServer;
	bBackupAct				: BOOL;
	bWritePersisAct			: BOOL;
	bWOCDisabled			: BOOL;
	eErrorID				: E_BACnet_Error;
END_VAR
VAR
	{region 'General'}
		nUpdateCount	 	: UDINT := 0;
	{endregion}
	{region 'Object List'}
		{attribute 'hide'}
		ipFirstObject		: I_BACnet_BaseObject;
		{attribute 'hide'}
		ipLastObject		: I_BACnet_BaseObject;
		{attribute 'hide'}
		nObjectCount		: UDINT;
	{endregion}
	{region 'Interface Pointer'}
		{attribute 'hide'}
		oServerOID			: OTCID; 
		{attribute 'hide'}
		iServer 			: ITcIoBACnetPlcServer;
		{attribute 'hide'}
		iDevice				: ITcIoBACnetPlcDevice;
		{attribute 'hide'}
		oDeviceOID			: OTCID;
		{attribute 'hide'}
		iObject				: ITcIoBACnetPlcObject;
	{endregion}
	{region 'Internal'}
		_ObjectId			: DWORD;	
		_ServerStatus		: WORD;
		_ServerControl		: WORD;
		_fbWritePersistent	: FB_WritePersistentData	:= (PORT:=TwinCAT_SystemInfoVarList._AppInfo.AdsPort, TMOUT:=T#1S, MODE:=E_PersistentMode.SPDM_2PASS);
		_rtrigBackup		: R_TRIG;
		_rtrigReset			: R_TRIG;
		_rtrigWritePers		: R_TRIG;
		_ePersDataState		: E_BACnet_PersistentDataState;
		_nPlcPort			: T_AmsPort;
		_tCyclicWrPers		: TON;
	{endregion}
	{region 'Misc'}
		{attribute 'hide'}
		fbLogMsg			: FB_BA_LogMessage;
	{endregion}
	{region 'Temporary'}
		_hResult			: HRESULT;
	{endregion}
END_VAR

IF (__ISVALIDREF(Adapter)) THEN
	Adapter();
END_IF
// Remind current number of update counter:
nUpdateCount := Adapter._nUpdateCount;

CASE (eState) OF
	E_BACnet_ServerState.eInitServer:
		eErrorID := E_BACnet_Error.eNoError;
		
		// Check if NetID is plausible:
		IF (Adapter.sAmsNetId = '') THEN
			fbLogMsg.Show1(ADSLOG_MSGTYPE_ERROR, 'D20', 'Configured AMS-NetID "%s" is invalid!', F_STRINGEx(Adapter.sAmsNetId), FALSE);
			eErrorID := E_BACnet_Error.eNoValidNetId;
		ELSIF (Adapter.eDevState <= E_BACnet_AdapterStatus.eInit) THEN
			; // Wait for adapter to get initialized.
		ELSIF (iDevice = 0) THEN
			Reset();
			iDevice := Adapter.Device;
			IF (iDevice <> 0) THEN
				iDevice.TcAddRef();
				iDevice.GetDeviceData(ADR(TwinCAT_SystemInfoVarList._AppInfo.ObjId), SIZEOF(OTCID), E_BACnet_DeviceData.eSetPlcOID);
			END_IF
		END_IF
		
		IF (iServer = 0) THEN
			IF (iDevice <> 0) THEN
				_hResult := iDevice.GetClientById(16#FFFFFFFF, ADR(iServer));
			ELSIF (oServerOID <> 0) THEN
				_hResult := FW_ObjMgr_GetObjectInstance(oid:=oServerOID, iid:=TC_GLOBAL_IID_LIST.IID_ITcIoBACnetPlcServer, pipUnk:=ADR(iServer));
			ELSE
				_hResult := S_OK;
			END_IF
			IF (iServer <> 0) THEN
				_hResult := iServer.GetAdsPort(ADR(tAmsPort));
				
				// Get Device-Object:
				IF (SUCCEEDED(_hResult)) THEN
					_hResult := iServer.GetObjectByObjectId(ADR(iObject), 16#23FFFFF);
					IF (SUCCEEDED(_hResult)) THEN
						_hResult := SEL(ReadPropertyUDInt(E_BACnetPropIdentifier.PropObjectIdentifier, _ObjectId), E_FAIL, S_OK);
					END_IF
					IF (SUCCEEDED(_hResult)) THEN
						_hResult := iObject.GetPropertyValue(E_BACnetPropIdentifier.PropProtocolRevision, ADR(nRev), 0);
					END_IF
					eErrorID := SEL(SUCCEEDED(_hResult), E_BACnet_Error.eInvalidServer, E_BACnet_Error.eNoError);
				END_IF
				
				// Indicate stack begin of object initialization: 
				_hResult := iServer.OnPlcAction(E_BACnet_PlcAction.eStart);
				IF (SUCCEEDED(_hResult)) THEN
					oDeviceOID := iServer.GetBACnetDeviceOid();
					IF (oDeviceOID = 0) THEN
						fbLogMsg.Show(ADSLOG_MSGTYPE_ERROR, 'D47', 'Internal error!', FALSE);
						eErrorID:=E_BACnet_Error.eInvalidServer;
					ELSE
						FW_ObjMgr_GetObjectInstance(oid:=oDeviceOID, iid:=TC_GLOBAL_IID_LIST.IID_ITcIoBACnetPlcDevice, pipUnk:=ADR(iDevice));
						
						// Start initializing objects:
						eState := E_BACnet_ServerState.eInitDefObjs;
					END_IF
				ELSE
					IF (iDevice = 0) THEN
						eErrorID := E_BACnet_Error.eInvalidTask;
						fbLogMsg.Show(ADSLOG_MSGTYPE_ERROR, 'D56', 'Task configuration invalid!', FALSE);
					ELSE
						fbLogMsg.Show1(ADSLOG_MSGTYPE_ERROR, 'D60', 'Internal error "0x%x"!', F_DINT(_hResult), FALSE);
						eErrorID := E_BACnet_Error.eInvalidServer;
					END_IF
					FW_SafeRelease(ADR(iServer));
					iServer:=0;				
				END_IF
			ELSE
				IF (_hResult = S_OK) THEN
					; // Resolving server...
				ELSE
					eErrorID := E_BACnet_Error.eInvalidServer;
					CASE (F_BACnet_FilterErrCode(_hResult)) OF
						E_AdsErr.DEVICE_NOTFOUND:
							fbLogMsg.Show(ADSLOG_MSGTYPE_ERROR, 'D74', 'BACnet-Server configuration missing!', FALSE);
					ELSE
						fbLogMsg.Show1(ADSLOG_MSGTYPE_ERROR, 'D78', 'BACnet-Server configuration invalid (Result: "0x%x")!', F_DINT(_hResult), FALSE);
					END_CASE
				END_IF
			END_IF
		END_IF
		
	E_BACnet_ServerState.eInitDefObjs:
		// [Hint] Initialization of defined objects DONE at this step.
		eState := E_BACnet_ServerState.eInitUndefObjs;
	
	E_BACnet_ServerState.eInitUndefObjs:
		// [Hint] Initialization of undefined objects DONE at this step.
		eState := E_BACnet_ServerState.eInitDefRefObjs;
	
	E_BACnet_ServerState.eInitDefRefObjs:
		// [Hint] Initialization of referring, defined objects DONE at this step.
		eState := E_BACnet_ServerState.eInitUndefRefObjs;
	
	E_BACnet_ServerState.eInitUndefRefObjs:
		// [Hint] Initialization of referring, undefined objects DONE at this step.
		
		_hResult := iServer.OnPlcAction(E_BACnet_PlcAction.eCreateFinish);
		IF (NOT SUCCEEDED(_hResult)) THEN
			fbLogMsg.Show1(ADSLOG_MSGTYPE_ERROR, 'D82', 'Internal error "0x%x"!', F_DINT(_hResult), FALSE);
			eErrorID := E_BACnet_Error.eInvalidServer;
		ELSIF (NOT Valid) THEN
			fbLogMsg.Show(ADSLOG_MSGTYPE_ERROR, 'D85', 'Invalid Server parameters!', FALSE);
			eErrorID := E_BACnet_Error.eInvalidParameter;
		ELSE
			// Validate user settings:
			IF (NOT F_BACnet_IsSchedBTypeValid(BACnet_Param.eSched_BType)) THEN
				fbLogMsg.Show(ADSLOG_MSGTYPE_ERROR, 'S90', 'Global parameter "eSchedB_Type" is invalid!', FALSE);
			END_IF
	
			eState := E_BACnet_ServerState.eOperation;
		END_IF
	
	E_BACnet_ServerState.eOperation:
		// Read properties:
		ReadPropertyInt(E_BACnetPropIdentifier.PropSystemStatus, eSysStatus);
		ReadPropertyInt(E_BACnetPropIdentifier.PropPersistentData, _ePersDataState);
		
		// Refresh server state:
		iServer.UpdateDeviceStatus(ADR(_ServerControl), ADR(_ServerStatus));
		bWOCDisabled := ((_ServerStatus AND 16#0004) = 16#0004);

		// Backup (Trigger writing of persistent data):
		_rtrigWritePers(CLK := bWritePersistent);
		_tCyclicWrPers(IN := (NOT _fbWritePersistent.BUSY), PT := tWritePersistent);
		
		IF (_fbWritePersistent.START) THEN
			IF (NOT _fbWritePersistent.BUSY) THEN
				// Writing persistent data finished:
				_ServerControl.1 := TRUE;
				_fbWritePersistent.START := FALSE;
			END_IF
		ELSE
			_ServerControl.1 := FALSE;
			_fbWritePersistent.START :=
				(eSysStatus = E_BACnet_DeviceStatus.eBackupInProgress) OR_ELSE
				(_ePersDataState = E_BACnet_PersistentDataState.eWrite) OR_ELSE
				(_rtrigWritePers.Q) OR_ELSE
				(_tCyclicWrPers.Q);
		END_IF
		_fbWritePersistent(BUSY=>bBackupAct);
		
	E_BACnet_ServerState.Invalid:
		;
		
ELSE
	fbLogMsg.Show1(ADSLOG_MSGTYPE_ERROR, 'S100', 'Invalid server state "%d"!', F_BYTE(eState), FALSE);
	eErrorID := E_BACnet_Error.eInvalidParameter;
END_CASE

IF (Error) THEN
	IF (eState = E_BACnet_ServerState.Invalid) THEN
		// Error occured in past cycles.
		
		// Reset Trigger:
		_rtrigReset(CLK:=bReset);
		IF (_rtrigReset.Q) OR_ELSE ((eErrorID < E_BACnet_Error.FirstResetError) OR (eErrorID >= E_BACnet_Error.LastResetError)) THEN
			_rtrigReset(CLK:=FALSE);
			Reset();
		END_IF
	ELSE
		// Error occured this cycle.
		Reset();
		eState := E_BACnet_ServerState.Invalid;
	END_IF
END_IF

// Control:
_ServerControl.2 := bDisableWOC;		// Disable write-on-change
_ServerControl.11 := Operational;		// PLC running - process data valid

{attribute 'hide'}
METHOD GetObjectByID : BOOL
VAR_INPUT
	tObjectID	: T_BACnet_ObjectIdentifier;
END_VAR
VAR_OUTPUT
	iResult		: I_BACnet_BaseObject;
END_VAR
iResult := ipFirstObject;
WHILE (iResult <> 0) DO
	IF (iResult.ObjectID = tObjectID) THEN
		GetObjectByID := TRUE;
		RETURN;
	END_IF
	iResult := iResult.NextObject;
END_WHILE
END_METHOD

{attribute 'hide'}
METHOD RegisterObject : BOOL
VAR_INPUT
	iObject	  : I_BACnet_BaseObject;
END_VAR
IF (iObject <> 0) THEN
	IF (nObjectCount = 0) THEN
		ipFirstObject := iObject;
	ELSE
		ipLastObject.NextObject := iObject;
	END_IF
	ipLastObject := iObject;
	nObjectCount := (nObjectCount + 1);
	
	RegisterObject := TRUE;
END_IF
END_METHOD

{attribute 'hide'}
PROPERTY ObjectCount : UDINT
GET
VAR
	cnt : UDINT;
END_VAR
IF iObject = 0 THEN
	ObjectCount:=0;
	RETURN;
END_IF

IF S_OK = iObject.SyncReadProperty(E_BACnetPropIdentifier.PropObjectList, ADR(cnt), 0, 0) THEN
 	ObjectCount:=cnt;
	RETURN;
END_IF

ObjectCount:=0;
END_GET
END_PROPERTY

{attribute 'hide'}
PROPERTY ServerItf : ITcIoBACnetPlcServer
GET
ServerItf := iServer;
END_GET
END_PROPERTY

METHOD PRIVATE Reset
IF iServer <> 0 THEN
	iServer.OnPlcAction(E_BACnet_PlcAction.eSuspend); // SUSPEND - delete all pointers to PLC
	FW_SafeRelease(ADR(iServer));
	iServer:=0;
END_IF
IF iObject <> 0 THEN
	FW_SafeRelease(ADR(iObject));
	iObject:=0;
END_IF	
IF iDevice <> 0 THEN
	FW_SafeRelease(ADR(iDevice));
	iDevice:=0;
END_IF 

// Object List:
ipLastObject := 0;
nObjectCount := 0;

eState := E_BACnet_ServerState.eInitServer;
eSysStatus := E_BACnet_DeviceStatus.Invalid;
bWOCDisabled := FALSE;
END_METHOD

// Called after online change.
{attribute 'call_after_online_change_slot' := '10'}
METHOD PROTECTED OnPostOnlineChange
Reset();
END_METHOD

PROPERTY Error : BOOL
GET
Error := (eErrorID <> E_BACnet_Error.eNoError);
END_GET
END_PROPERTY

PROPERTY Operational : BOOL
GET
Operational := (eState=E_BACnet_ServerState.eOperation);
END_GET
END_PROPERTY

PROPERTY Valid : BOOL
GET
Valid := (_ObjectId <> 16#00000000);
END_GET
END_PROPERTY

{attribute 'hide'}
METHOD ReadPropertyInt : BOOL
VAR_INPUT
	ePropID : E_BACnetPropIdentifier;
	value : REFERENCE TO INT;
END_VAR
VAR_STAT
	_hr : HRESULT;
	_val : DINT;
	_size : DINT := SIZEOF(_val);
END_VAR
IF iObject<>0 AND (__ISVALIDREF(value)) THEN
	_hr:=iObject.SyncReadProperty(TO_INT(ePropID), ADR(_val), ADR(_size), 16#FFFFFFFF);
	IF (_hr = S_OK) THEN
		value := TO_INT(_val);
		ReadPropertyInt:=TRUE;
		RETURN;
	END_IF
END_IF
ReadPropertyInt:=FALSE;
END_METHOD

{attribute 'hide'}
METHOD ReadPropertyUDInt : BOOL
VAR_INPUT
	ePropID : E_BACnetPropIdentifier;
	value : REFERENCE TO UDINT;
END_VAR
VAR
	_hr : HRESULT;
	_size : DINT := 4;
END_VAR
IF iObject<>0 AND (__ISVALIDREF(value)) THEN
	_hr:=iObject.SyncReadProperty(TO_INT(ePropID), ADR(value), ADR(_size), 16#FFFFFFFF);
	IF (_hr = S_OK) THEN
		ReadPropertyUDInt:=TRUE;
		RETURN;
	END_IF
END_IF
ReadPropertyUDInt:=FALSE;
END_METHOD

METHOD FB_Exit : BOOL
VAR_INPUT
	 bInCopyCode : BOOL; // if TRUE, the exit method is called for exiting an instance that is copied afterwards (online change).
END_VAR
Reset();
END_METHOD

END_FUNCTION_BLOCK

// POUs/Helper/[internal]/F_BACnet_FilterErrCode
{attribute 'hide'}
FUNCTION F_BACnet_FilterErrCode : HRESULT
VAR_INPUT
	hResult		: HRESULT;
END_VAR

F_BACnet_FilterErrCode := TO_UINT(hResult) AND 16#FFF;

END_FUNCTION

// POUs/Helper/[internal]/Validation-Functions/F_BACnet_IsSchedBTypeValid
{attribute 'hide'}
FUNCTION F_BACnet_IsSchedBTypeValid : BOOL
VAR_INPUT
	eType		: E_BACnet_SchedBType;
END_VAR

F_BACnet_IsSchedBTypeValid := ((E_BACnet_SchedBType.First <= eType) AND_THEN (eType <= E_BACnet_SchedBType.Last));

END_FUNCTION

// TEST/TestPackage/BACKUP
PROGRAM BACKUP
VAR
	cfgTsZip	: FB_BACnet_File := (bEnBackupFile:=TRUE, sObjectName := 'CurrentConfig.tszip',	sFileName := 'CurrentConfig.tszip');
	plcBootdata : FB_BACnet_File := (bEnBackupFile:=TRUE, sObjectName := 'Port_851.bootdata', 	sFileName := 'Plc\Port_851.bootdata');
	plcApp 		: FB_BACnet_File := (bEnBackupFile:=TRUE, sObjectName := 'Port_851.app', 		sFileName := 'Plc\Port_851.app');
	plcCrc 		: FB_BACnet_File := (bEnBackupFile:=TRUE, sObjectName := 'Port_851.crc', 		sFileName := 'Plc\Port_851.crc');
	plcTiZip	: FB_BACnet_File := (bEnBackupFile:=TRUE, sObjectName := 'Port_851_boot.tizip', sFileName := 'Plc\Port_851_boot.tizip');
END_VAR

cfgTsZip();
plcBootdata();
plcApp();
plcCrc();
plcTiZip();

END_PROGRAM

// POUs/Local/Objects/FB_BACnet_File
// File Object
{attribute 'enable_dynamic_creation'}
FUNCTION_BLOCK FB_BACnet_File EXTENDS FB_BACnet_Object
VAR_INPUT CONSTANT 
	{region 'Fixed Parameters'}
		{attribute 'parameterCategory':='General'}
		bEnBackupFile : BOOL;
		{attribute 'parameterCategory':='General'}
		{attribute 'TcEncoding':='UTF-8'}
		sFileName : T_MaxString;
	{endregion}
END_VAR
VAR_INPUT CONSTANT PERSISTENT
	{attribute 'parameterCategory':='General'}
	bArchive : BOOL;	 
	{attribute 'parameterCategory':='General'}
	bReadOnly : BOOL;	 	 
END_VAR
VAR_OUTPUT
	nFileSize		: UDINT;
END_VAR

SUPER^();

METHOD PROTECTED OnObjectStateChanged
SUPER^.OnObjectStateChanged();

CASE (tState) OF
	TCOM_STATE.TCOM_STATE_PREOP:
		// SyncHandler:
		RequestSyncHandlers(3, 2);
		
		IF (sFileName <> '') THEN
			RequestSyncHandlers(0, 1);
			WritePropertyString(E_BACnetPropIdentifier.PropFileName, sFileName);
			EnableProperty(E_BACnetPropIdentifier.PropFileName, TRUE);
			WriteProtectProperty(E_BACnetPropIdentifier.PropFileName, TRUE);
		END_IF
		IF (bEnBackupFile) THEN
			WritePropertyString(E_BACnetPropIdentifier.PropFileType, 'TwinCAT Configuration File');
		END_IF
		
	TCOM_STATE.TCOM_STATE_SAFEOP:
		;
	
	TCOM_STATE.TCOM_STATE_OP:
		SyncProperty(E_BACnetPropIdentifier.PropArchive, SIZEOF(bArchive), ADR(bArchive), 0, eFullSync_InitPLC);
		SyncProperty(E_BACnetPropIdentifier.PropReadOnly, SIZEOF(bReadOnly), ADR(bReadOnly), 0, eFullSync_InitPLC);
		SyncProperty(E_BACnetPropIdentifier.PropFileSize, SIZEOF(nFileSize), ADR(nFileSize), 0, eSync_FromSupplement);
		IF (sFileName <> '') THEN
			SyncProperty(E_BACnetPropIdentifier.PropFileName, SIZEOF(sFileName), ADR(sFileName), 0, eSync_ToSupplement);
		END_IF
		
END_CASE
END_METHOD

METHOD FB_init : BOOL
VAR_INPUT
	bInitRetains : BOOL; // if TRUE, the retain variables are initialized (warm start / cold start)
	bInCopyCode : BOOL;  // if TRUE, the instance afterwards gets moved into the copy code (online change)
END_VAR
eObjectType := E_BACnetObjType.ObjFile;
END_METHOD

END_FUNCTION_BLOCK

// POUs/Local/Objects/[Base]/Basic/FB_BACnet_Object
{attribute 'reflection'}
FUNCTION_BLOCK ABSTRACT FB_BACnet_Object EXTENDS FB_BACnet_BaseObject IMPLEMENTS I_BACnet_Object, I_BACnet_ObjectOwner
VAR_INPUT CONSTANT PERSISTENT
	{region 'Variable Parameters'}
		{attribute 'parameterCategory':='General'}
		{attribute 'TcEncoding':='UTF-8'}
		sObjectName : T_MaxString;
		{attribute 'parameterCategory':='General'}
		{attribute 'TcEncoding':='UTF-8'}
		sDescription : T_MaxString;
	{endregion}
END_VAR
VAR
	{region 'UserInit'}
		iParent						: I_BACnet_View;
	{endregion}
END_VAR
VAR
	{region 'COV'}
		bObjNameChanged				: BOOL;
		bDescriptionChanged			: BOOL;
	{endregion}
	{region 'General'}
		{attribute 'instance-path'}
		{attribute 'no_init'}
		sSymbolPath  				: T_MaxString;														// Full symbol path of current instance
		sSymbolName  				: STRING;															// Symbol name of current instance
	{endregion}
	{region 'Linked Object-List'
		{attribute 'hide'}
		iPrevSibling				: I_BACnet_Object;
		{attribute 'hide'}
		iNextSibling				: I_BACnet_Object;
	{endregion}
	{region 'Internal'}
		{attribute 'hide'}
		bParentInit					: BOOL := TRUE;
		{attribute 'hide'}
		fbLogMsg					: FB_BA_LogMessage;
	{endregion}
END_VAR
VAR CONSTANT
	{region 'Payload-Balancing'}
		{attribute 'hide'}
		COV_UPDATE_CYCLE			: UDINT	:= 100;														// Execute COV-indication every X cycles to ALL properties
		{attribute 'hide'}
		COV_UPDATE_SPLIT			: UDINT	:= 100;														// Splits all objects in max. X groups to execute COV-indication
	{endregion}
END_VAR

IF (bReady) THEN
	// Request COV-Update:
	bUpdateCOV := (nUpdateCount MOD COV_UPDATE_CYCLE) = (nObjectInstance MOD COV_UPDATE_SPLIT);
	
	SUPER^();
	
	IF (iParent <> 0) AND_THEN (iParent.Ready) THEN
		// Concatenate changed titles at runtime:
		ValidateTitles();
	END_IF
	
ELSE
	SUPER^();
	IF (bReady) THEN
		OnPostInit();
	END_IF
END_IF

// Unused - Implemented for compatibility reason!
{attribute 'hide'}
METHOD OnBACnetObjectStateChanged
VAR_INPUT
	tState			: TCOM_STATE;
END_VAR
END_METHOD

{attribute 'hide'}
METHOD OnCycle : BOOL
VAR_INPUT
	bUpdateCOV		: BOOL;
END_VAR
// Call current instance directly (Without using an external 'UpdateCOV' implementation):
THIS^();
END_METHOD

METHOD INTERNAL RemoveFromLinkedObjList
VAR_IN_OUT
	iFirstChild			: I_BACnet_Object;
	iLastChild			: I_BACnet_Object;
END_VAR
VAR
	_iThisObj			: I_BACnet_Object;
END_VAR
_iThisObj := THIS^;

// Remove current instance from linked object list:
IF (iFirstChild = _iThisObj) THEN
	// Current instance is at first index position:
	iFirstChild := NextSibling;
	
ELSIF (PrevSibling <> 0) THEN
	// Current instance is not at first index position:
	PrevSibling.NextSibling := NextSibling;
END_IF

IF (NextSibling = 0) THEN
	// Current instance is at last index position:
	iLastChild := PrevSibling;
ELSE
	// Current instance is not at last index position:
	NextSibling.PrevSibling := PrevSibling;
END_IF
END_METHOD

{attribute 'suppress_wrn_C0410'}
{attribute 'hide'}
PROPERTY LogMsg : REFERENCE TO FB_BA_LogMessage
GET
LogMsg REF= fbLogMsg;
END_GET
END_PROPERTY

{attribute 'hide'}
PROPERTY NextSibling : I_BACnet_Object
GET
NextSibling := iNextSibling;
END_GET
SET
iNextSibling := NextSibling;
END_SET
END_PROPERTY

{attribute 'hide'}
PROPERTY PrevSibling : I_BACnet_Object
GET
PrevSibling := iPrevSibling;
END_GET
SET
iPrevSibling := PrevSibling;
END_SET
END_PROPERTY

{attribute 'hide'}
PROPERTY SymbolName : POINTER TO STRING
GET
SymbolName := ADR(sSymbolName);
END_GET
END_PROPERTY

{attribute 'hide'}
PROPERTY SymbolPath : POINTER TO T_MaxString
GET
SymbolPath := ADR(sSymbolPath);
END_GET
END_PROPERTY

// Unused - Implemented for compatibility reason!
{attribute 'hide'}
METHOD Close
iPrevSibling := 0;
iNextSibling := 0;

SUPER^.Close();
END_METHOD

METHOD INTERNAL DynamicInit : BOOL
VAR_INPUT
	fbProducer			: POINTER TO FB_BACnet_DynObjectManager;
	nObjectInstance		: UDINT;
	sObjectName			: T_MaxString;
	sDescription		: T_MaxString;
	fbParent			: POINTER TO FB_BACnet_View		:= 0;
END_VAR
IF (fbProducer <> 0) THEN
	// Init current instance:
	THIS^.fbDynProducer := fbProducer;
	THIS^.nObjectInstance := nObjectInstance;
	THIS^.sObjectName := sObjectName;
	THIS^.sDescription := sDescription;
	
	// Remove concatenation command if existing:
	F_BA_RemovePrefix(sObjectName, BACnet_Globals.sCmd_ConcatTitle);
		
	sSymbolName := sObjectName;
	
	IF (fbParent = 0) THEN
		sSymbolPath := CONCAT('_dynamic.', sObjectName);
	ELSE
		sSymbolPath := CONCAT(fbParent^.sSymbolPath, '.');
		sSymbolPath := CONCAT(sSymbolPath, sObjectName);
		
		iParent := fbParent^;
	END_IF
	
	// Call current instance once:
	// > Necessary for parents to get their children registered!
	THIS^();
	
	DynamicInit := NOT Error;
END_IF
END_METHOD

METHOD PROTECTED OnObjectStateChanged
SUPER^.OnObjectStateChanged();

CASE (tState) OF
	TCOM_STATE.TCOM_STATE_PREOP:
		// Ensure UTF-8 Encoding:
		F_BA_EnsureUTF8(ADR(sObjectName), SIZEOF(sObjectName));
		F_BA_EnsureUTF8(ADR(sDescription), SIZEOF(sDescription));
	
		// SyncHandler:
		RequestSyncHandlers(2, 3);
		
		IF (iParent <> 0) THEN
			// Register current instance into parent:
			__QUERYPOINTER(iParent, _fbView);
			_fbView^.AddObject(THIS^);
		END_IF

	TCOM_STATE.TCOM_STATE_SAFEOP:
		;
		
	TCOM_STATE.TCOM_STATE_OP:
		// Build titles:
		bObjNameChanged := TRUE;
		bDescriptionChanged := TRUE;
		
		ValidateTitles();
		
		IF S_OK <> SyncProperty(E_BACnetPropIdentifier.PropObjectName, SIZEOF(sObjectName), ADR(sObjectName), ADR(bObjNameChanged), eFullSync_InitPLC) THEN
			// Init object name failed!
			// > Try init symbol path instead:
			_hResult := SyncProperty(E_BACnetPropIdentifier.PropObjectName, SIZEOF(sSymbolPath), ADR(sSymbolPath), 0, eSync_ToSupplement);
			IF _hResult = S_OK THEN
				fbLogMsg.Show1(ADSLOG_MSGTYPE_ERROR, 'OOSC26', 'Duplicate use of object name "%s"! Applied symbolname instead of objectname.', F_STRING(sObjectName), FALSE);
				sObjectName := sSymbolPath;
			ELSE
				fbLogMsg.Show2(ADSLOG_MSGTYPE_ERROR, 'OOSC29', 'Failed to initialize object name of "%s" (Error: 0x%x)!', F_STRING(sSymbolPath), F_DINT(_hResult), FALSE);
			END_IF
		END_IF
		
		SyncProperty(E_BACnetPropIdentifier.PropDescription, SIZEOF(sDescription), ADR(sDescription), ADR(bDescriptionChanged), eFullSync_InitPLC);
		
END_CASE
END_METHOD

// Called on first operational cycle after initialization.
METHOD PROTECTED OnPostInit
END_METHOD

METHOD INTERNAL ValidateReference : BOOL
VAR_IN_OUT
	iReference			: I_BACnet_Object;
	tIdentifier			: T_BACnet_ObjectIdentifier;
END_VAR
VAR_INPUT
	eExpectedType		: E_BACnetObjType				:= 16#FF;
END_VAR
VAR
	_bIdentifierValid	: BOOL;
	_iObject			: I_BACnet_BaseObject;
	_iRef				: I_BACnet_Object;
END_VAR
_bIdentifierValid := F_BACnet_IsObjIdentifierValid(tIdentifier);

IF (NOT Ready) THEN
	// Ignore (may persistent stored) pointers:
	iReference := 0;
END_IF
IF (NOT _bIdentifierValid) AND (iReference = 0) THEN
	// Reference undefined:
	ValidateReference := TRUE;
ELSE
	IF (NOT _bIdentifierValid) AND_THEN (iReference <> 0) THEN
		// Interface-pointer of object exists:
		// > Get Object-Identifier:
		tIdentifier := iReference.ObjectID;
		
	ELSIF (_bIdentifierValid) THEN
		// Object identifier of object exists:
		// > Get Interface-pointer:
		IF (Server.GetObjectByID(tIdentifier, iResult=>_iObject)) AND_THEN (__QUERYINTERFACE(_iObject, _iRef)) THEN
			iReference := _iRef;
		ELSE
			tIdentifier := BACnet_Globals.nBACnetObjId_None;
		END_IF
	END_IF
	
	IF (tIdentifier = BACnet_Globals.nBACnetObjId_None) OR (iReference = 0) THEN
		fbLogMsg.Show1(ADSLOG_MSGTYPE_ERROR, 'VOI15', 'Resolving referred object "%d" failed!', F_DWORD(tIdentifier), TRUE);
		
	ELSIF (eExpectedType <> 16#FF) AND_THEN (iReference.ObjectType <> eExpectedType) THEN
		fbLogMsg.Show1(ADSLOG_MSGTYPE_ERROR, 'VOI20', 'Validation of object "%d" failed: type unexpected!', F_DWORD(tIdentifier), TRUE);
			
	ELSE
		// Ensure initialized (And than referrable!) reference:
		IF (NOT iReference.Ready) AND_THEN (__QUERYPOINTER(iReference, _fbObject)) THEN
			// Call referred object for initialization:
			_fbObject^();
		END_IF
	
		ValidateReference := TRUE;
		RETURN;
	END_IF
	
	tIdentifier := 0;
	iReference := 0;
END_IF
END_METHOD

METHOD PROTECTED ConcatTitle : BOOL
VAR_IN_OUT
	sInstTitle			: T_MaxString;
END_VAR
VAR_INPUT
	sParentTitle		: T_MaxString;
	sSeparator			: STRING;
END_VAR
VAR
	iConcatLen			: INT;
END_VAR
iConcatLen := LEN(BACnet_Globals.sCmd_ConcatTitle);

IF (LEFT(sInstTitle, iConcatLen) = BACnet_Globals.sCmd_ConcatTitle) THEN
	// Remove concatenation-command:
	sInstTitle := DELETE(sInstTitle, iConcatLen, 1);
	
	IF (sParentTitle <> '') THEN
		// Concatenate parent title:
		sInstTitle := CONCAT(sSeparator, sInstTitle);
		sInstTitle := CONCAT(sParentTitle, sInstTitle);
	END_IF
END_IF
END_METHOD

METHOD PROTECTED ValidateTitles
// Concatenate titles at runtime:
IF bObjNameChanged THEN
	bObjNameChanged := FALSE;
	ConcatTitle(sObjectName, SEL((iParent <> 0), '', iParent.ObjectName), BACnet_Param.sSeparator_ObjectName);
END_IF
IF bDescriptionChanged THEN
	bDescriptionChanged := FALSE;
	ConcatTitle(sDescription, SEL((iParent <> 0), '', iParent.Description), BACnet_Param.sSeparator_Description);
END_IF
END_METHOD

PROPERTY Parent : I_BACnet_View
GET
Parent := iParent;
END_GET
SET
IF (iParent = 0) THEN
	iParent := Parent;
ELSE
	IF (Parent <> 0) THEN
		fbLogMsg.Show(ADSLOG_MSGTYPE_ERROR, 'P4', 'Object already assigned to parent!', FALSE);
	END_IF
END_IF
END_SET
END_PROPERTY

METHOD ReadPropertyExceptionSched : HRESULT
VAR_IN_OUT
	aCalendar			: ARRAY[*] OF ST_BACnet_SchedCalendar;
	aException			: ARRAY[*] OF ST_BACnet_SchedException;
END_VAR
VAR_INPUT
	eDatatype			: E_BACnet_ValueChoice;
END_VAR
VAR
	_i					: INT;
END_VAR
ReadPropertyExceptionSched := SUPER^.ReadPropertyExceptionSched(aCalendar, aException, eDatatype);

IF (ReadPropertyExceptionSched = S_OK) THEN
	// Validate referred objects:
	FOR _i := 1 TO BACnet_Param.nSched_CalendarCount DO
		ValidateReference(aCalendar[_i].iRefCalendar, aCalendar[_i].tRefCalendarID, E_BACnetObjType.ObjCalendar);
	END_FOR
END_IF
END_METHOD

METHOD ReadPropertyReference : HRESULT
VAR_INPUT
	eProperty				: E_BACnetPropIdentifier;
END_VAR
VAR_IN_OUT
	stRefObject				: ST_BACnet_ObjectPropertyReference;
END_VAR
ReadPropertyReference := SUPER^.ReadPropertyReference(eProperty, stRefObject);

IF (ReadPropertyReference = S_OK) THEN
	ValidateReference(stRefObject.iObject, stRefObject.tObjectID, 16#FF);
END_IF
END_METHOD

METHOD WritePropertyExceptionSched : HRESULT
VAR_IN_OUT
	aCalendar			: ARRAY[*] OF ST_BACnet_SchedCalendar;
	aException			: ARRAY[*] OF ST_BACnet_SchedException;
END_VAR
VAR_INPUT
	eDatatype			: E_BACnet_ValueChoice;
END_VAR
VAR
	_i					: INT;
END_VAR
// Validate referred objects:
FOR _i := 1 TO BACnet_Param.nSched_CalendarCount DO
	ValidateReference(aCalendar[_i].iRefCalendar, aCalendar[_i].tRefCalendarID, E_BACnetObjType.ObjCalendar);
END_FOR

WritePropertyExceptionSched := SUPER^.WritePropertyExceptionSched(aCalendar, aException, eDatatype);
END_METHOD

METHOD WritePropertyReference : HRESULT
VAR_INPUT
	eProperty				: E_BACnetPropIdentifier;
END_VAR
VAR_IN_OUT
	stReference				: ST_BACnet_ObjectPropertyReference;
END_VAR
ValidateReference(stReference.iObject, stReference.tObjectID, 16#FF);

WritePropertyReference := SUPER^.WritePropertyReference(eProperty, stReference);
END_METHOD

PROPERTY Description : T_MaxString
GET
Description := sDescription;
END_GET
SET
sDescription := Description;
END_SET
END_PROPERTY

PROPERTY ObjectName : T_MaxString
GET
ObjectName := sObjectName;
END_GET
SET
sObjectName := ObjectName;
END_SET
END_PROPERTY

METHOD FB_init : BOOL
VAR_INPUT
	bInitRetains : BOOL; // if TRUE, the retain variables are initialized (warm start / cold start)
	bInCopyCode : BOOL;  // if TRUE, the instance afterwards gets moved into the copy code (online change)
END_VAR
iOwner := THIS^;

IF (bInitRetains) THEN
	// Remove "Solution Project" title:
	sSymbolPath := right(sSymbolPath, len(sSymbolPath)-find(sSymbolPath,'.'));
	// Remove "PLC Project" title:
	// sSymbolPath := right(sSymbolPath, len(sSymbolPath)-find(sSymbolPath,'.'));
END_IF
	
sSymbolName := F_BA_StringRight(sSymbolPath, '.');
	
fbLogMsg.Path := sSymbolPath;

// Indicate inheritance of project structure as default:
sObjectName := CONCAT(BACnet_Globals.sCmd_ConcatTitle, sSymbolName);
END_METHOD

END_FUNCTION_BLOCK

// POUs/Local/Objects/[Internal]/FB_BACnet_BaseObject
{attribute 'enable_dynamic_creation'}
{attribute 'no_assign'}
{attribute 'hide'}
FUNCTION_BLOCK FB_BACnet_BaseObject IMPLEMENTS I_BACnet_BaseObject
VAR_INPUT CONSTANT
	{region 'Fixed Parameters'}
		{attribute 'parameterCategory':='General'}
		{attribute 'no_copy'}
		Server : REFERENCE TO FB_BACnet_Server := BACnet_Globals.DefaultServer;
	{endregion}
END_VAR
VAR_INPUT CONSTANT PERSISTENT
	{region 'Fixed Parameters'}
		{attribute 'parameterCategory':='General'}
		nObjectInstance : UDINT := BACnet_Globals.nBACnetInstId_Auto;
	{endregion}
END_VAR
VAR
	{region 'Output-Properties'}
		bReady						: BOOL;
	{endregion}
	{region 'SubInit'}
		eObjectType					: E_BACnetObjType				:= 16#FFFF;
		{attribute 'hide'}
		iOwner						: I_BACnet_ObjectOwner;												// Owner of current Instance (Pointer to current instance per default)
	{endregion}
END_VAR
VAR
	{region 'General'}
		tState						: TCOM_STATE					:= TCOM_STATE.TCOM_STATE_INIT;
		eErrorID					: E_BACnet_Error				:= E_BACnet_Error.eNoError;
		tObjectID					: T_BACnet_ObjectIdentifier		:= BACnet_Globals.nBACnetObjId_None;
		bUpdateCOV					: BOOL;
			 
		{attribute 'conditionalshow'}
		nCycPropCnt					: DINT;
		{attribute 'conditionalshow'}
		aSyncHandlers				: ARRAY [E_BA_SyncMode.eFromSupplement .. E_BA_SyncMode.eToSupplement] OF UDINT;
			 
		{attribute 'conditionalshow'}
		nPlcSync					: DINT;
	{endregion}
	{region 'Interface Pointer'}
		{attribute 'conditionalshow'}
		ipSrv						: ITcIoBACnetPlcServer;
		{attribute 'conditionalshow'}
		ipObj						: ITcIoBACnetPlcObject;
	{endregion}
	{region 'Object List'}
		{attribute 'hide'}
		ipNextObject				: I_BACnet_BaseObject;
		{attribute 'hide'}
		bIsRegistered				: BOOL;
	{endregion}
	{region 'Internal'}
		{attribute 'hide'}
		bIsReused					: BOOL;																// Object was already created in BACnet stack.
		{attribute 'hide'}
		nUpdateCount 				: UDINT := 0;
		{attribute 'conditionalshow'}
		aReqSyncHandlers			: ARRAY [E_BA_SyncMode.eFromSupplement .. E_BA_SyncMode.eToSupplement] OF UDINT;
		{attribute 'hide'}
		{attribute 'no_copy'}
		fbDynProducer				: POINTER TO FB_BACnet_DynObjectManager;							// Pointer to producing manager, if dynamically created.
	{endregion}
END_VAR
VAR_STAT
	{region 'Temporary'}
		{attribute 'hide'}
		_fbObject					: POINTER TO FB_BACnet_Object;
		{attribute 'hide'}
		_fbView						: POINTER TO FB_BACnet_View;
		{attribute 'hide'}
		_sSymbolPath				: T_MaxString;
		{attribute 'hide'}
		_hResult 					: HRESULT;
		{attribute 'hide'}
		_i							: E_BA_SyncMode;
		{attribute 'hide'}
		_nSize						: DINT;
		{attribute 'hide'}
		_nTemp						: UDINT;
		{attribute 'hide'}
		_tObjID						: T_BACnet_ObjectIdentifier;
		{attribute 'hide'}
		_ipPlcObj					: ITcIoBACnetPlcObject;
	{endregion}	
END_VAR

// Update device:
IF (Server.nUpdateCount = nUpdateCount) THEN
	Server();
END_IF
// Remind current number of update counter:
nUpdateCount := Server.nUpdateCount;

IF (Error) THEN
	bReady := FALSE;
ELSE
	CASE (Server.eState) OF
		E_BACnet_ServerState.eInitServer:
			; // Wait for server to get initialized.
			
		E_BACnet_ServerState.eInitDefObjs,
		E_BACnet_ServerState.eInitUndefObjs,
		E_BACnet_ServerState.eInitDefRefObjs,
		E_BACnet_ServerState.eInitUndefRefObjs:
			// Wait for appropriate server state to initialize current instance:
			IF (NOT bReady) AND_THEN (IsInitReady()) THEN
				bReady := FALSE;
	
				IF (iOwner = 0) THEN
					eErrorID := E_BACnet_Error.eInvalidParameter;
					iOwner.LogMsg.Show(ADSLOG_MSGTYPE_ERROR, 'O23', 'Owner of BACnet object not defined!', FALSE);
				ELSIF (nObjectInstance > BACnet_Globals.nBACnetInstId_Auto) THEN
					eErrorID := E_BACnet_Error.eInvalidObjectId;
					_nTemp := (BACnet_Globals.nBACnetInstId_Auto-1);
					iOwner.LogMsg.Show2(ADSLOG_MSGTYPE_ERROR, 'O28', 'Creating object failed due to invalid instance ID %d! (Valid range: 0 - %d)', F_UDINT(nObjectInstance), F_UDINT(_nTemp), FALSE);
				ELSE
					ipSrv := Server.ServerItf;
					IF (ipSrv <> 0) THEN
						IF (eObjectType = E_BACnetObjType.ObjDevice) THEN
							_hResult := ipSrv.GetObjectByObjectId(ADR(ipObj), 16#23FFFFF);
							IF (_hResult = S_OK) THEN
								State := TCOM_STATE.TCOM_STATE_PREOP;
								bIsReused := TRUE;
							END_IF
						ELSE
							tObjectID := F_BACnet_GetObjId(eObjectType, nObjectInstance);
							
							_sSymbolPath := iOwner.SymbolPath^;
							_hResult := ipSrv.GetObjectBySymbolName(ADR(ipObj), _sSymbolPath, LEN(_sSymbolPath));
							IF (_hResult = S_OK) THEN
								_nSize := SIZEOF(_tObjID);
								_hResult := ipObj.GetPropertyValue(E_BACnetPropIdentifier.PropObjectIdentifier, ADR(_tObjID), ADR(_nSize));
								IF (_hResult = S_OK) THEN
									// Check PLC object for changed properties within live time of the stack object:
									IF (eObjectType <> F_BACnet_GetObjType(_tObjID)) THEN
										// Object type has changed:
										_hResult := E_FAIL;
									ELSIF (nObjectInstance <> F_BACnet_GetObjInstance(_tObjID)) AND (nObjectInstance <> BACnet_Globals.nBACnetInstId_Auto) THEN
										// Object instance has changed:
										_hResult := E_FAIL;
									END_IF
									
									IF (_hResult <> S_OK) THEN
										// Delete old (now unused) stack-object.
										ipSrv.DeletePlcObjectRT(ADR(ipObj));
										ipObj := 0;
									END_IF
								END_IF
								
								IF (_hResult = S_OK) THEN
									// Continue using existing BACnet-Object:
									bIsReused := TRUE;
									State := TCOM_STATE.TCOM_STATE_PREOP;
									_hResult := S_OK;
								END_IF
							END_IF
							
							IF (_hResult <> S_OK) THEN
								// BACnet-Object hast to be created:
								// > Check for existing objects in stack that are already using the current Instance-ID.
								IF (ipSrv.GetObjectByObjectId(ADR(ipObj), tObjectID) = S_OK) THEN
									IF (Server.GetObjectByID(tObjectID)) THEN
										eErrorID := E_BACnet_Error.eDuplicateObjectId;
										ipObj := 0;
										
										iOwner.LogMsg.Show1(ADSLOG_MSGTYPE_ERROR, 'O42', 'Creating object failed due to duplicated use of instance ID "%d"!', F_UDINT(nObjectInstance), FALSE);
										_hResult := S_OK;
									ELSE
										// The existing object is not used by another PLC object at this time!
										// > Delete the existing stack object before creating a new stack-object for this instance:
										ipSrv.DeletePlcObjectRT(ADR(ipObj));
										ipObj := 0;
									END_IF
								END_IF
							END_IF
										
							IF (_hResult <> S_OK) THEN
								// Create new BACnet-Object:
								_hResult := ipSrv.CreatePlcObjectRT(ADR(ipObj), eObjectType, nObjectInstance, TCOM_STATE.TCOM_STATE_PREOP);
								IF (_hResult = S_OK) THEN
									// Init basic properties:
									ipObj.SyncWriteProperty(E_BACnetPropIdentifier.PropPlcSymbolName, ADR(_sSymbolPath), LEN(_sSymbolPath), 16#FFFFFFFF);
							
									State := TCOM_STATE.TCOM_STATE_PREOP;
							
									// Apply requested number of SyncHandlers:
									ApplySyncHandler();
								
									_hResult := ipSrv.CreatePlcObjectRT(ADR(ipObj), eObjectType, nObjectInstance, TCOM_STATE.TCOM_STATE_OP);
									IF _hResult <> S_OK THEN
										eErrorID := E_BACnet_Error.eCreateObject;
										iOwner.LogMsg.Show1(ADSLOG_MSGTYPE_ERROR, 'O82', 'Creating object failed! (Error 0x%x)', F_DINT(_hResult), FALSE);
									END_IF
								ELSE
									eErrorID := E_BACnet_Error.eCreateObject;
									iOwner.LogMsg.Show2(ADSLOG_MSGTYPE_ERROR, 'O86', 'Creating object failed! (Instance: "%d", Error: 0x%x)', F_UDINT(nObjectInstance), F_DINT(_hResult), FALSE);			
								END_IF
							END_IF
							
							IF (IsDynamic) THEN
								; // No need to register dynamically created objects into server.
							ELSE
								// Register current instance in server:
								IF (NOT Server.RegisterObject(THIS^)) THEN
									iOwner.LogMsg.Show(ADSLOG_MSGTYPE_ERROR, 'O20', 'Failed to register current instance in internal object list!', FALSE);	
								END_IF
							END_IF
						END_IF
					END_IF
				END_IF
			END_IF
		
		E_BACnet_ServerState.eOperation:
			IF (bReady) THEN
				// Instance operational.
				
				// Set number of properties to be synchronized in current cycle:
				nPlcSync := SEL(bUpdateCOV, nCycPropCnt, 255);
			ELSIF (ipObj = 0) THEN
				eErrorID := E_BACnet_Error.eCreateObject;
				iOwner.LogMsg.Show1(ADSLOG_MSGTYPE_ERROR, 'O120', 'Creating object timed out! (Instance: "%d")', F_UDINT(nObjectInstance), FALSE);
			ELSE
				// Complete object initialization:
				State := TCOM_STATE.TCOM_STATE_SAFEOP;
				
				bReady := (NOT Error);
				State := TCOM_STATE.TCOM_STATE_OP;
				
				// SyncHandler-Diagnose:
				{IF defined (Debug_LogReqSyncHandler)}
					// Define max. difference from "Requested" to "Applied":
					{IF hasvalue(Debug_LogReqSyncHandler,'Suspect')}
						_nSize := 3;
					{ELSE}
						_nSize := 0;
					{END_IF}
					IF (MAX(F_BA_DifferenceDINT(TO_DINT(aReqSyncHandlers[E_BA_SyncMode.eFromSupplement]), TO_DINT(aSyncHandlers[E_BA_SyncMode.eFromSupplement])),
						F_BA_DifferenceDINT(TO_DINT(aReqSyncHandlers[E_BA_SyncMode.eToSupplement]), TO_DINT(aSyncHandlers[E_BA_SyncMode.eToSupplement]))) > _nSize) THEN

						iOwner.LogMsg.Show4(ADSLOG_MSGTYPE_HINT, 'DEBUG.O134', '[SyncHandlers] Requested: %d/%d, Applied: %d/%d (from/to)',
											F_UDINT(aReqSyncHandlers[E_BA_SyncMode.eFromSupplement]), F_UDINT(aReqSyncHandlers[E_BA_SyncMode.eToSupplement]),
											F_UDINT(aSyncHandlers[E_BA_SyncMode.eFromSupplement]), F_UDINT(aSyncHandlers[E_BA_SyncMode.eToSupplement]),
											FALSE);	
					END_IF
				{ELSE}
					IF (NOT bIsReused) THEN
						IF (aSyncHandlers[E_BA_SyncMode.eFromSupplement] > aReqSyncHandlers[E_BA_SyncMode.eFromSupplement]) OR
							(aSyncHandlers[E_BA_SyncMode.eToSupplement] > aReqSyncHandlers[E_BA_SyncMode.eToSupplement]) THEN
							iOwner.LogMsg.Show4(ADSLOG_MSGTYPE_WARN, 'O142', 'Inconsistent SyncHandlers! Requested: %d/%d, Applied: %d/%d (from/to)',
												F_UDINT(aReqSyncHandlers[E_BA_SyncMode.eFromSupplement]), F_UDINT(aReqSyncHandlers[E_BA_SyncMode.eToSupplement]),
												F_UDINT(aSyncHandlers[E_BA_SyncMode.eFromSupplement]), F_UDINT(aSyncHandlers[E_BA_SyncMode.eToSupplement]),
												FALSE);	
						END_IF
					END_IF
				{END_IF}
						  
				bReady := NOT Error;
			END_IF
			
	END_CASE
END_IF

// Unused - Implemented for compatibility reason!
{attribute 'hide'}
METHOD OnCycle : BOOL
VAR_INPUT
	bUpdateCOV		: BOOL;
END_VAR
THIS^.bUpdateCOV := bUpdateCOV;

THIS^();

OnCycle := NOT Error;
END_METHOD

{attribute 'hide'}
PROPERTY NextObject : I_BACnet_BaseObject
GET
NextObject := ipNextObject;
END_GET
SET
ipNextObject := NextObject;
END_SET
END_PROPERTY

{attribute 'hide'}
METHOD View_AddSubordinate : BOOL
VAR_INPUT
	iObject			: I_BACnet_BaseObject;
END_VAR
VAR
	_fbObject		: POINTER TO FB_BACnet_BaseObject;
	_sTemp			: T_MaxString;
	_listEntry		: ST_BACnetRaw_DeviceObjectReference;
END_VAR
IF (iObject = 0) THEN
	F_BA_LogMessage(ADSLOG_MSGTYPE_ERROR, 'RCO05', 'Undefined object!');
	
ELSIF (eObjectType <> E_BACnetObjType.ObjStructuredView) THEN
	F_BA_LogMessage(ADSLOG_MSGTYPE_ERROR, 'RCO02', 'Invalid object type!');
	
ELSIF (NOT __QUERYPOINTER(iObject, _fbObject)) THEN
	F_BA_LogMessage(ADSLOG_MSGTYPE_ERROR, 'RCO08', 'Cast of object-interface failed!');
	
ELSE
	_listEntry.tObjId := iObject.ObjectID;
			
	AddPropertyElementPtr(E_BACnetPropIdentifier.PropSubordinateList, ADR(_listEntry), SIZEOF(_listEntry));

	// (BETA) ... "PropSubordinateAnnotations"
	// > Kann hier das 'ReadPropertyString()' wirklich eingespart werden?? Weil das ja intern UTF8-dekodiert..!?
	(*
	IF (_fbObject^.ReadPropertyString(E_BACnetPropIdentifier.PropObjectname, _sTemp)) THEN
		AddPropertyElementString(E_BACnetPropIdentifier.PropSubordinateAnnotations, _sTemp);
	END_IF
	*)
	
	// Register child-object in current instance (Called "Subordinate" in BACnet):
	_sTemp := _fbObject^.iOwner.SymbolName^;
	AddPropertyElement(E_BACnetPropIdentifier.PropSubordinateAnnotations, _sTemp);

	View_AddSubordinate := TRUE;
END_IF
END_METHOD

{attribute 'hide'}
METHOD View_RemoveSubordinate : BOOL
VAR_INPUT
	iObject			: I_BACnet_BaseObject;
END_VAR
IF (iObject = 0) THEN
	F_BA_LogMessage(ADSLOG_MSGTYPE_ERROR, 'RCO05', 'Undefined object!');
	
ELSIF (eObjectType <> E_BACnetObjType.ObjStructuredView) THEN
	F_BA_LogMessage(ADSLOG_MSGTYPE_ERROR, 'RCO02', 'Invalid object type!');
	
ELSE
	

	// (BETA) ...
	// TODO



	View_RemoveSubordinate := TRUE;
END_IF
END_METHOD

// Unused - Implemented for compatibility reason!
{attribute 'hide'}
METHOD Close
IF ipObj <> 0 THEN
	FW_SafeRelease(ADR(ipObj));
	ipObj:=0;
END_IF

ipSrv := 0;
tState := 0;

FOR _i := E_BA_SyncMode.eFromSupplement TO E_BA_SyncMode.eToSupplement DO
	aSyncHandlers[_i] := 0;
	aReqSyncHandlers[_i] := 0;
END_FOR

// Object List:
ipNextObject := 0;
bIsRegistered := FALSE;

fbDynProducer := 0;

bIsReused := FALSE;
bReady := FALSE;
END_METHOD

METHOD PRIVATE Sched_ReadEntry : BOOL
VAR_INPUT
	eExpectedType	: E_BACnet_ValueChoice;
	pTimeValue		: POINTER TO ST_BACnet_TimeValueList;
	pEntry			: POINTER TO ST_BA_SchedEntry;
END_VAR
IF (pTimeValue = 0) OR_ELSE (pEntry = 0) THEN
	iOwner.LogMsg.Show(ADSLOG_MSGTYPE_WARN, 'SRE02', 'Invalid time value', TRUE);
	
ELSIF (pTimeValue^.nEntrySize = 0) THEN
	Sched_ReadEntry := FALSE;
	
ELSIF (pTimeValue^.stListEntry.stValue.eValueChoice <> E_BACnet_ValueChoice.eNullValue) AND (pTimeValue^.stListEntry.stValue.eValueChoice <> eExpectedType) THEN
	iOwner.LogMsg.Show1(ADSLOG_MSGTYPE_WARN, 'SRE04', 'Invalid time value type "%d"!', F_INT(pTimeValue^.stListEntry.stValue.eValueChoice), TRUE);
	
ELSE
	CASE (pTimeValue^.stListEntry.stValue.eValueChoice) OF
		E_BACnet_ValueChoice.eNullValue:
			pEntry^.eState := E_BA_SchedEntryState.eNull;
			
		E_BACnet_ValueChoice.eEnumerationValue:
			pEntry^.eState := E_BA_SchedEntryState.eValue;
			MEMCPY(ADR(pEntry^.uValue), ADR(pTimeValue^.stListEntry.stValue.stValue.nEnumValue), pTimeValue^.stListEntry.stValue.nSize - SIZEOF(pTimeValue^.stListEntry.stValue.stValue.eChoice));
			
	ELSE
		pEntry^.eState := E_BA_SchedEntryState.eValue;
		MEMCPY(ADR(pEntry^.uValue), ADR(pTimeValue^.stListEntry.stValue.stValue), pTimeValue^.stListEntry.stValue.nSize);
	END_CASE
	
	pEntry^.stTime := pTimeValue^.stListEntry.stTime;
	Sched_ReadEntry := TRUE;
END_IF
END_METHOD

METHOD PRIVATE Sched_SetNextDay : BOOL
VAR_IN_OUT
	_pDailySched					: POINTER TO ST_BACnet_DailySchedule;
	_cbTmpSize						: UDINT;
	_cbTotalBuf						: UDINT;
	_pOldTimeValue					: POINTER TO ST_BACnet_TimeValueList;
	_nDayTmp						: DINT;
	_nDayEntryTmp					: DINT;
	_pTimeValue						: POINTER TO ST_BACnet_TimeValueList;
END_VAR
IF eObjectType = E_BACnetObjType.ObjSchedule THEN
	Sched_SetNextDay := ((_pDailySched^.nEntrySize AND 16#80000000) = 16#80000000);
	
	_cbTmpSize := F_BACnet_AlignedSize(_pDailySched^.nEntrySize AND 16#7FFFFFFF) + SIZEOF(_pDailySched^.nEntrySize) + SIZEOF(_pDailySched^.nRes);
	_pDailySched := _pDailySched + _cbTmpSize;
	_cbTotalBuf := _cbTotalBuf + _cbTmpSize;
	_pOldTimeValue := 0;
	_nDayEntryTmp := 1;
	
	IF Sched_SetNextDay THEN
		_pTimeValue := ADR(_pDailySched^.stListEntry);
		_nDayTmp := _nDayTmp + 1;
	END_IF
END_IF
END_METHOD

METHOD PRIVATE Sched_SetNextTimeVal : BOOL
VAR_IN_OUT
	_pDailySched					: POINTER TO ST_BACnet_DailySchedule;
	_pTimeValue						: POINTER TO ST_BACnet_TimeValueList;
	_cbTmpSize						: UDINT;
	_pOldTimeValue					: POINTER TO ST_BACnet_TimeValueList;
END_VAR
IF eObjectType = E_BACnetObjType.ObjSchedule THEN
	Sched_SetNextTimeVal := (_pTimeValue^.nEntrySize AND 16#80000000) = 16#80000000;
	
	_cbTmpSize := F_BACnet_AlignedSize(_pTimeValue^.nEntrySize AND 16#7FFFFFFF) + SIZEOF(_pDailySched^.stListEntry.nEntrySize) + SIZEOF(_pDailySched^.stListEntry.nRes);
	_pOldTimeValue := _pTimeValue;
	_pTimeValue := _pTimeValue + _cbTmpSize;
END_IF
END_METHOD

METHOD PRIVATE Sched_WriteEntry : BOOL
VAR_INPUT
	eValueChoice 	: E_BACnet_ValueChoice;
	pTimeValue		: POINTER TO ST_BACnet_TimeValueList;
	pEntry 			: POINTER TO ST_BA_SchedEntry;
END_VAR
CASE (pEntry^.eState) OF
	E_BA_SchedEntryState.eNull:
		pTimeValue^.stListEntry.stValue.nSize := 0;
		eValueChoice := E_BACnet_ValueChoice.eNullValue;
		
	E_BA_SchedEntryState.eValue:
		CASE (eValueChoice) OF
			E_BACnet_ValueChoice.eBoolValue:
				pTimeValue^.stListEntry.stValue.nSize := SIZEOF(pEntry^.uValue.bVal);
				
			E_BACnet_ValueChoice.eEnumerationValue:
				pTimeValue^.stListEntry.stValue.nSize := SIZEOF(UDINT) + SIZEOF(E_BACnet_EnumerationValueChoice);
				
			E_BACnet_ValueChoice.eRealValue:
				pTimeValue^.stListEntry.stValue.nSize := SIZEOF(pEntry^.uValue.rVal);
				
			E_BACnet_ValueChoice.eUnsignedValue:
				pTimeValue^.stListEntry.stValue.nSize := SIZEOF(pEntry^.uValue.udiVal);
				
		ELSE
			iOwner.LogMsg.Show(ADSLOG_MSGTYPE_WARN, 'SWE20', 'Unsupported data type!', TRUE);
			RETURN;
		END_CASE
ELSE
	iOwner.LogMsg.Show1(ADSLOG_MSGTYPE_WARN, 'SWE24', 'Unsupported exception scheduler pEntry type "%d"!', F_INT(pEntry^.eState), TRUE);
	RETURN;
END_CASE
		
// Set data:
pTimeValue^.stListEntry.stTime := pEntry^.stTime;
IF pTimeValue^.stListEntry.stTime.nReserve = 255 AND pTimeValue^.stListEntry.stTime.nHour <> 255 THEN
	pTimeValue^.stListEntry.stTime.nReserve:=0;
END_IF
pTimeValue^.stListEntry.stValue.eValueChoice := eValueChoice;
pTimeValue^.stListEntry.stValue.nRes1 := 0;
IF eValueChoice = E_BACnet_ValueChoice.eEnumerationValue THEN
	pTimeValue^.stListEntry.stValue.stValue.eChoice := E_BACnet_EnumerationValueChoice.eBinaryPV;
	pTimeValue^.stListEntry.stValue.stValue.nEnumValue := TO_UDINT(pEntry^.uValue.bVal);
ELSE
	pTimeValue^.stListEntry.stValue.nRes1 := 0;					
	MEMCPY(ADR(pTimeValue^.stListEntry.stValue.stValue), ADR(pEntry^.uValue), pTimeValue^.stListEntry.stValue.nSize);						
END_IF
	
// Calculate time-value pEntry size:
pTimeValue^.nEntrySize := pTimeValue^.stListEntry.stValue.nSize
						+ SIZEOF(pTimeValue^.stListEntry.nRes)
						+ SIZEOF(pTimeValue^.stListEntry.stTime)
						+ SIZEOF(pTimeValue^.stListEntry.stValue.eValueChoice)
						+ SIZEOF(pTimeValue^.stListEntry.stValue.nRes1)
						+ SIZEOF(pTimeValue^.stListEntry.stValue.nSize);
END_METHOD

METHOD PRIVATE DeleteObject : BOOL
IF (ipObj <> 0) AND (ipSrv <> 0) THEN
	IF S_OK <> ipSrv.DeletePlcObjectRT(ADR(ipObj)) THEN
		RETURN;
	END_IF
END_IF 

ipObj := 0;
ipSrv := 0;
eErrorID := E_BACnet_Error.eNoError;

DeleteObject := TRUE;
END_METHOD

METHOD PRIVATE IsInitReady : BOOL
// Check condition:
CASE (eObjectType) OF
	E_BACnetObjType.ObjCommand,
	E_BACnetObjType.ObjEventEnrollment,
	E_BACnetObjType.ObjSchedule,
	E_BACnetObjType.ObjAveraging,
	E_BACnetObjType.ObjTrendLog,
	E_BACnetObjType.ObjPulseConverter,
	E_BACnetObjType.ObjTrendLogMultiple:
		// Current instance can refer objects.
		// Assume an initialized reference-object in "E_BACnet_ServerState.eInit[...]RefObjs" state.
		IF (Server.eState < E_BACnet_ServerState.eInitDefRefObjs) THEN
			RETURN;
		END_IF
END_CASE

// Wait for appropriate state to start initialization:
CASE (Server.eState) OF
	E_BACnet_ServerState.eInitDefObjs,
	E_BACnet_ServerState.eInitDefRefObjs:
		IsInitReady := (nObjectInstance<>BACnet_Globals.nBACnetInstId_Auto);
	E_BACnet_ServerState.eInitUndefObjs,
	E_BACnet_ServerState.eInitUndefRefObjs:
		IsInitReady := (nObjectInstance=BACnet_Globals.nBACnetInstId_Auto);
END_CASE
END_METHOD

METHOD PROTECTED OnObjectStateChanged
CASE (tState) OF
	TCOM_STATE.TCOM_STATE_PREOP:
		// [Hint] To be done in this step:
		// - Disable properties
		// - Initialization of property-memory (e.g. Buffer Size)
		// - Set max. property count via "SetPropertyCount()"
		
		ipObj.GetPropertyValue(E_BACnetPropIdentifier.PropObjectIdentifier, ADR(tObjectID), 0);
		nObjectInstance := F_BACnet_GetObjInstance(tObjectID);
	
		// SyncHandler:
		RequestSyncHandlers(0, 1);
		
	TCOM_STATE.TCOM_STATE_SAFEOP:
		// [Hint] To be done in this step:
		// - Initialize property-sync to important (means COV-indication) properties
		
		SyncProperty(E_BACnetPropIdentifier.PropPlcUpdateTrigger, SIZEOF(nPlcSync), ADR(nPlcSync), 0, eSync_ToSupplement);
		
		// Get Object-ID:
		ipObj.GetPropertyValue(E_BACnetPropIdentifier.PropObjectIdentifier, ADR(tObjectID), 0);
		
	TCOM_STATE.TCOM_STATE_OP:
		// [Hint] To be done in this step:
		// - Write protection of properties
		// - Init Entry Count of Arrays: SyncWrite(pData:=Null, nData:=0)
		// - Init Entry Count of Lists: SyncWrite(pData:=ADR(bByteArray), nData:=8)		// -> 'bByteArray' has to be init with NULL
		
		// [Hint] Keep in mind:
		// - Initialize "Resolution" beforce other referring properties are initialized. 
		//   E.g. "COV-Increment"
		// - Register COV-Notification via "SyncProperty(X, Y, Z, bHasChanged, S)":
		//   The trigger variable "bHasChanged" will indicate a COV when if the synchronized property has been written from inside the PLC via "WriteProperty()"-methods.
		
END_CASE

// Notify owner:
iOwner.OnBACnetObjectStateChanged(tState);
END_METHOD

// Called after online change.
{attribute 'call_after_online_change_slot' := '10'}
METHOD PROTECTED OnPostOnlineChange
Close();
END_METHOD

METHOD Acknowledge : BOOL
VAR_INPUT
	eTransition			: E_BA_EventTransition	:= E_BA_EventTransition.Invalid;
	sMessage			: STRING				:= '';
END_VAR
VAR
	nAckEvent			: UDINT;
END_VAR
IF (Ready) THEN
	CASE (eTransition) OF
		E_BA_EventTransition.eToOffnormal:
			F_BACnet_SetBitFieldBit(ADR(nAckEvent), 2);
		E_BA_EventTransition.eToFault:
			F_BACnet_SetBitFieldBit(ADR(nAckEvent), 1);
		E_BA_EventTransition.eToNormal:
			F_BACnet_SetBitFieldBit(ADR(nAckEvent), 0);
	ELSE
		// Acknowledge all events:
		nAckEvent := 16#FFFFFFFF;
	END_CASE
	
	Acknowledge := (ipObj.SyncAckTransition(TO_UINT(nAckEvent), sMessage, TO_INT(LEN(sMessage))) = S_OK);
END_IF
END_METHOD

PROPERTY Error : BOOL
GET
Error := (eErrorID <> E_BACnet_Error.eNoError);
END_GET
END_PROPERTY

PROPERTY IsDynamic : BOOL
GET
IsDynamic := (fbDynProducer <> 0);
END_GET
END_PROPERTY

PROPERTY ObjectID : T_BACnet_ObjectIdentifier
GET
ObjectID := tObjectID;
END_GET
END_PROPERTY

PROPERTY ObjectInstance : UDINT
GET
ObjectInstance := nObjectInstance;
END_GET
END_PROPERTY

PROPERTY ObjectType : E_BACnetObjType
GET
ObjectType := eObjectType;
END_GET
END_PROPERTY

PROPERTY Ready : BOOL
GET
Ready := bReady;
END_GET
END_PROPERTY

PROPERTY State : TCOM_STATE
GET
State := tState;
END_GET
SET
PROTECTED
VAR
	_bSetSyncHand	: BOOL;
END_VAR
IF tState <> State THEN
	tState := State;
	OnObjectStateChanged();
END_IF
END_SET
END_PROPERTY

METHOD EnableProperty : HRESULT
VAR_INPUT
	eID : E_BACnetPropIdentifier;
	bEnable : BOOL := TRUE;
END_VAR
EnableProperty := ipObj.SyncPropertyState(eID, bEnable);
END_METHOD

METHOD SetPropertyCount : BOOL
VAR_INPUT
	nCount			: UDINT;
	eSyncMode		: E_BA_SyncMode;
END_VAR
VAR CONSTANT
	LIMIT_MIN		: UDINT		:= 43;
END_VAR
IF (bIsReused) THEN
	// Count already set!
ELSE
	CASE (eSyncMode) OF
		E_BA_SyncMode.eFromSupplement:
			_hResult := WritePropertyUDInt(E_BACnetPropIdentifier.PropCyclicInMaxCfg, nCount);
		E_BA_SyncMode.eToSupplement:
			_hResult := WritePropertyUDInt(E_BACnetPropIdentifier.PropCyclicOutMaxCfg, nCount);
	ELSE
		iOwner.LogMsg.Show(ADSLOG_MSGTYPE_ERROR, 'SPC23', 'Invalid Sync-Mode defined!', TRUE);
		RETURN;
	END_CASE
	
	IF _hResult = S_OK THEN
		SetPropertyCount := TRUE;
	ELSE
		iOwner.LogMsg.Show1(ADSLOG_MSGTYPE_ERROR, 'SPC20', 'Failed to set property count! (Error 0x%x)', F_DINT(_hResult), TRUE);
	END_IF
END_IF
END_METHOD

METHOD WriteProtectProperty : HRESULT
VAR_INPUT
	eID : E_BACnetPropIdentifier;
	bProtect : BOOL := TRUE;
END_VAR
WriteProtectProperty := ipObj.SyncPropertyProtection(eID, bProtect);
END_METHOD

METHOD AddPropertyElement : BOOL
VAR_INPUT
	eProperty : E_BACnetPropIdentifier;
	xValue : ANY;
END_VAR
VAR
	_stData : POINTER TO ST_BACnet_ValueList;
	_pData : PVOID;
	_nSize : UDINT;
END_VAR
IF (ipObj <> 0) AND_THEN (bReady) THEN
	CASE (xValue.TypeClass) OF
		__SYSTEM.TYPE_CLASS.TYPE_STRING:
			AddPropertyElement := (F_BACnet_EncodeUTF8(xValue.pValue, TO_UDINT(xValue.diSize), ADR(BACnet_Globals.aDefaultBuffer), SIZEOF(BACnet_Globals.aDefaultBuffer), _nSize) <> 0);
			IF (AddPropertyElement) THEN
				_pData := ADR(BACnet_Globals.aDefaultBuffer);
			END_IF
			
	ELSE
		iOwner.LogMsg.Show2(ADSLOG_MSGTYPE_ERROR, 'APE10', 'Unimplemented datatype of property "%d"! (Type class "%d")', F_INT(eProperty), F_DWORD(xValue.TypeClass), TRUE);
		RETURN;
	END_CASE
	
	IF (AddPropertyElement) THEN
		_hResult := ipObj.SyncWriteProperty(TO_INT(eProperty), _pData, TO_UINT(F_BACnet_AlignedSize(_nSize)), 16#FFFFFFFE);

		IF (_hResult <> S_OK) THEN
			AddPropertyElement := FALSE;
			_hResult := F_BACnet_FilterErrCode(_hResult);
			
			CASE (eProperty) OF
				E_BACnetPropIdentifier.PropSubordinateAnnotations:
					IF (_hResult = TO_DINT(E_AdsErr.DEVICE_ACCESSDENIED)) THEN
						iOwner.LogMsg.Show(ADSLOG_MSGTYPE_ERROR, 'APE25', 'Insufficient memory (LIST_ALLOC_MEM_BYTES, MAX_PROPERTY_ARRAYELEMENTS) to register in subordinate list!', FALSE);
						RETURN;
					END_IF
			END_CASE
			
			iOwner.LogMsg.Show2(ADSLOG_MSGTYPE_ERROR, 'APE20', 'Writing element to property "%d" failed! (Error: 0x%x)', F_INT(eProperty), F_DINT(_hResult), TRUE);
		END_IF
	ELSE
		iOwner.LogMsg.Show1(ADSLOG_MSGTYPE_ERROR, 'APE23', 'Failed to prepare element of property "%d"!', F_INT(eProperty), TRUE);
	END_IF
END_IF
END_METHOD

METHOD AddPropertyElementPtr : BOOL
VAR_INPUT
	ePropID : E_BACnetPropIdentifier;
	pData : PVOID;
	nData : UINT;
END_VAR
VAR
	_cbResult : UDINT;
END_VAR
IF (ipObj <> 0) AND_THEN (bReady) THEN
	_hResult := ipObj.SyncWriteProperty(TO_INT(ePropID), pData, nData, 16#FFFFFFFE);
	AddPropertyElementPtr:=(S_OK = _hResult);
END_IF
END_METHOD

METHOD RemoveArrayElements : BOOL
VAR_INPUT
	ePropID : E_BACnetPropIdentifier;
END_VAR
IF (ipObj <> 0) THEN
	_hResult := ipObj.SyncWriteProperty(ePropID, 0, 0, 16#FFFFFFFF);
	RemoveArrayElements := (S_OK=_hResult);
END_IF
END_METHOD

METHOD RemoveListElements : BOOL
VAR_INPUT
	ePropID : E_BACnetPropIdentifier;
END_VAR
VAR
	aData : ARRAY [0 .. 7] OF BYTE;
END_VAR
IF (ipObj <> 0) THEN
	_hResult := ipObj.SyncWriteProperty(ePropID, ADR(aData), SIZEOF(aData), 16#FFFFFFFF);
	RemoveListElements:=(S_OK = _hResult);
END_IF
END_METHOD

METHOD SetNumberOfStates : BOOL
VAR_INPUT
	nCount			: UDINT;
END_VAR
IF (ipObj <> 0) AND_THEN (nCount > 0) THEN
	_hResult := ipObj.SyncWriteProperty(E_BACnetPropIdentifier.PropNumberOfStates, ADR(nCount), SIZEOF(nCount), 16#FFFFFFFF);
	SetNumberOfStates:=(S_OK = _hResult);
END_IF
END_METHOD

METHOD ReadProperty : HRESULT
VAR_INPUT
	ePropID : E_BACnetPropIdentifier;
	pData : PVOID;
	nData : POINTER TO DINT;
END_VAR
VAR
	_size : DINT := 4;
END_VAR
IF (ipObj <> 0) AND (pData <> 0) AND (nData > 0) THEN
	ReadProperty := ipObj.SyncReadProperty(TO_INT(ePropID), pData, nData, 16#FFFFFFFF);

	IF (ReadProperty <> S_OK) THEN
		iOwner.LogMsg.Show2(ADSLOG_MSGTYPE_ERROR, 'RP5', 'Reading property "%d" failed (Error "0x%x")!', F_INT(ePropID), F_DINT(ReadProperty), TRUE);
	END_IF
ELSE
	ReadProperty := E_FAIL;
END_IF
END_METHOD

METHOD ReadPropertyAckedTransitions : HRESULT
VAR_INPUT
	value : REFERENCE TO ST_BA_EventTransitions;
END_VAR
VAR
	_flags : DWORD;
	_size : DINT := 2;
END_VAR
VAR CONSTANT
	ePropID : E_BACnetPropIdentifier := E_BACnetPropIdentifier.PropAckedTransitions;
END_VAR
IF (ipObj <> 0) AND (__ISVALIDREF(value)) THEN
	ReadPropertyAckedTransitions := ipObj.SyncReadProperty(TO_INT(ePropID), ADR(value), ADR(_size), 16#FFFFFFFF);
	
	IF ReadPropertyAckedTransitions = S_OK THEN
		value.bToNormal:= F_BACnet_IsBitFieldBitSet(_flags, E_BACnet_EventTransitionBits.eToNormal);
		value.bToFault:= F_BACnet_IsBitFieldBitSet(_flags, E_BACnet_EventTransitionBits.eToFault);
		value.bToOffnormal:= F_BACnet_IsBitFieldBitSet(_flags, E_BACnet_EventTransitionBits.eToOffnormal);
	END_IF
ELSE
	ReadPropertyAckedTransitions := E_FAIL;
END_IF
END_METHOD

METHOD ReadPropertyBool : HRESULT
VAR_INPUT
	ePropID : E_BACnetPropIdentifier;
	bValue : REFERENCE TO BOOL;
END_VAR
VAR
	_size : DINT := 1;
END_VAR
IF (ipObj <> 0) AND (__ISVALIDREF(bValue)) THEN
	ReadPropertyBool := ReadProperty(ePropID, ADR(bValue), ADR(_size));
ELSE
	ReadPropertyBool := E_FAIL;
END_IF
END_METHOD

METHOD ReadPropertyByte : HRESULT
VAR_INPUT
	ePropID : E_BACnetPropIdentifier;
	nValue : REFERENCE TO BYTE;
END_VAR
VAR
	_size : DINT := 4;
END_VAR
IF (ipObj <> 0) AND (__ISVALIDREF(nValue)) THEN
	ReadPropertyByte := ReadProperty(ePropID, ADR(nValue), ADR(_size));
ELSE
	ReadPropertyByte := E_FAIL;
END_IF
END_METHOD

METHOD ReadPropertyDateList : HRESULT
VAR_IN_OUT
	aDateList				: ARRAY[*] OF ST_BA_CalendarEntry;
END_VAR
VAR
	_i						: DINT;
	_nLength, _nCount		: DINT;
	_iIndex, _iMin, _iMax	: DINT;
	
	_stEntry				: POINTER TO ST_BACnet_CalendarEntry;
END_VAR
IF (ipObj = 0) THEN
	_hResult := E_FAIL;
ELSE
	_nLength := SIZEOF(BACnet_Globals.aDefaultBuffer);
	_hResult := ReadProperty(E_BACnetPropIdentifier.PropDateList, ADR(BACnet_Globals.aDefaultBuffer), ADR(_nLength));
	
	IF (SUCCEEDED(_hResult)) THEN
		// Clear content:
		MEMSET(aDateList, 0, TO_UDINT(F_BA_DateListSize(aDateList)));
		
		_nCount := (_nLength / SIZEOF(ST_BACnet_CalendarEntry));
		IF (_nCount > 0) THEN
			_iMin := LOWER_BOUND(aDateList, 1);
			_iMax := UPPER_BOUND(aDateList, 1);
			_nCount := MIN(_nCount, (_iMax-_iMin+1));
			
			_stEntry := ADR(BACnet_Globals.aDefaultBuffer);
			_iIndex := _iMin;
			FOR _i := 0 TO (_nCount-1) DO
				aDateList[_iIndex].eType := (_stEntry^.eEventChoice+1);
				aDateList[_iIndex].uDate := (_stEntry^.uCalEntry);
				
				_stEntry := (_stEntry+SIZEOF(ST_BACnet_CalendarEntry));
				_iIndex := (_iIndex+1);
			END_FOR
		END_IF
	END_IF
END_IF

ReadPropertyDateList := _hResult;
END_METHOD

METHOD ReadPropertyEventEnable : HRESULT
VAR CONSTANT
	ePropID : E_BACnetPropIdentifier := E_BACnetPropIdentifier.PropEventEnable;
END_VAR
VAR_INPUT
	value : REFERENCE TO ST_BA_EventTransitions;
END_VAR
VAR
	_flags : WORD := 16#0005;
	_size : DINT := 2;
END_VAR
IF (ipObj <> 0) AND (__ISVALIDREF(value)) THEN
	ReadPropertyEventEnable := ReadProperty(ePropID, ADR(_flags), ADR(_size));
	
	IF (ReadPropertyEventEnable = S_OK) THEN
		value.bToNormal := _flags.13;
		value.bToFault := _flags.14;
		value.bToOffnormal := _flags.15;
	END_IF
ELSE
	ReadPropertyEventEnable := E_FAIL;
END_IF
END_METHOD

METHOD ReadPropertyEventParameter : HRESULT
VAR_IN_OUT
	stEventParameter				: ST_BACnet_EventParameter;
END_VAR
VAR
	_nLength		: DINT;
END_VAR
IF (ipObj = 0) THEN
	_hResult := E_FAIL;
ELSE
	_nLength := SIZEOF(BACnet_Globals.aDefaultBuffer);
	_hResult := ReadProperty(E_BACnetPropIdentifier.PropEventParameters, ADR(BACnet_Globals.aDefaultBuffer), ADR(_nLength));
	
	IF (SUCCEEDED(_hResult)) THEN
		MEMCPY(ADR(stEventParameter), ADR(BACnet_Globals.aDefaultBuffer), TO_UDINT(_nLength)); // Copy event type and header Info
		stEventParameter.nArgSize := _nLength - 8;
	ELSE
		stEventParameter.eEventType := E_BACnet_EventType.Invalid;
	END_IF
END_IF

ReadPropertyEventParameter := _hResult;
END_METHOD

METHOD ReadPropertyEventState : HRESULT
VAR CONSTANT
	ePropID : E_BACnetPropIdentifier := E_BACnetPropIdentifier.PropEventState;
END_VAR
VAR_INPUT
	value : REFERENCE TO E_BACnet_EventState;
END_VAR
VAR
	_size : DINT := SIZEOF(E_BACnet_EventState);
END_VAR
IF (ipObj <> 0) AND (__ISVALIDREF(value)) THEN
	ReadPropertyEventState := ReadProperty(ePropID, ADR(value), ADR(_size));
ELSE
	ReadPropertyEventState := E_FAIL;
END_IF
END_METHOD

METHOD ReadPropertyEventTimeStamps : HRESULT
VAR CONSTANT
	ePropID : E_BACnetPropIdentifier := E_BACnetPropIdentifier.PropEventTimeStamps;
END_VAR
VAR_INPUT
	value : REFERENCE TO ST_BACnet_EventTimeStamps;
END_VAR
VAR
	_size : DINT := SIZEOF(ST_BACnet_EventTimeStamps);
END_VAR
IF (ipObj <> 0) AND (__ISVALIDREF(value)) THEN
	ReadPropertyEventTimeStamps := ReadProperty(ePropID, ADR(value), ADR(_size));
ELSE
	ReadPropertyEventTimeStamps := E_FAIL;
END_IF
END_METHOD

METHOD ReadPropertyExceptionSched : HRESULT
VAR_IN_OUT
	aCalendar					: ARRAY[*] OF ST_BACnet_SchedCalendar;
	aException					: ARRAY[*] OF ST_BACnet_SchedException;
END_VAR
VAR_INPUT
	eDatatype					: E_BACnet_ValueChoice;
END_VAR
VAR
	// General:
	nLenTmp						: UDINT;
	nLength						: DINT;
	
	_cbTmpSize					: UDINT;
	_cbTotalEntry				: UDINT;
	_cbTotalBuf					: UDINT;

	_pDailySched				: POINTER TO ST_BACnet_SpecialEventList;
	_pTimeValue					: POINTER TO ST_BACnet_TimeValueList;
	_nTimeValue					: DINT;
	_nCalEntry					: DINT := 1;
	_nExcEntry					: DINT := 1;
	_calObjId					: T_BACnet_ObjectIdentifier;
	
	_nMaxSchedEntryCount		: DINT;
	_nMaxCalCount				: DINT;
	_nMaxExcptCount				: DINT;
	
	// [Bug-Workaround]: Diese scheiss Firma 3S
	// Sched_ReadEntry(eDatatype, _pTimeValue, aCalendar[_nCalEntry].aEntry[_nTimeValue]);			// "...aEntry[_nTimeValue]" ist immer der Pointer auf "aEntry[1]" :(
	_pCalEntry			: POINTER TO ST_BA_SchedEntry;
	
	// [Bug-Workaround]: Diese scheiss Firma 3S
	// Sched_ReadEntry(eDatatype, _pTimeValue, aException[_nExcEntry].aEntry[_nTimeValue]);			// "...aEntry[_nTimeValue]" ist immer der Pointer auf "aEntry[1]" :(
	_pExceptEntry		: POINTER TO ST_BA_SchedEntry;
END_VAR
IF ipObj = 0 THEN
	_hResult := E_FAIL;	
ELSIF (eDataType = E_BACnet_ValueChoice.eNullValue) THEN
	iOwner.LogMsg.Show(ADSLOG_MSGTYPE_ERROR, 'RWS05', 'Invalid datatype!', TRUE);
	_hResult := E_FAIL;
ELSE
	nLength := SIZEOF(BACnet_Globals.aDefaultBuffer);
	_hResult := ReadProperty(E_BACnetPropIdentifier.PropExceptionSchedule, ADR(BACnet_Globals.aDefaultBuffer), ADR(nLength));
	
	IF (SUCCEEDED(_hResult)) AND (nLength > 8) THEN
		// Clear content:
		MEMSET(aCalendar, 0, TO_UDINT(F_BA_CalendarSchedSize(aCalendar)));
		MEMSET(aException, 0, TO_UDINT(F_BA_ExceptionSchedSize(aException)));
			
		// Point to first data:
		_pDailySched:= ADR(BACnet_Globals.aDefaultBuffer);
		
		_nMaxSchedEntryCount := BACnet_Param.nSched_EntryCount;
		_nMaxCalCount := UPPER_BOUND(aCalendar, 1);
		_nMaxExcptCount := UPPER_BOUND(aException, 1);
		
		WHILE _pDailySched <> 0 DO
			IF _pDailySched^.stEvent.eEventChoice = E_BACnet_SpecialEventChoice.eCalendarReference THEN
				IF (_nCalEntry <= _nMaxCalCount) THEN
					MEMCPY(ADR(_calObjId), ADR(_pDailySched^.stEvent.eCalEntryChoice), SIZEOF(_calObjId));
					aCalendar[_nCalEntry].tRefCalendarID := _calObjId;
					aCalendar[_nCalEntry].eEventPriority := TO_INT(_pDailySched^.stEvent.nEventPriority);
					
					_pTimeValue := F_BACnet_EndOf(_pDailySched, SIZEOF(ST_BACnet_SpecialEventList));
					_pCalEntry := ADR(aCalendar[_nCalEntry].aEntry[1]);
					_nTimeValue := 1;
					WHILE _pTimeValue <> 0 DO
						IF (_nTimeValue <= _nMaxSchedEntryCount) THEN
							Sched_ReadEntry(eDatatype, _pTimeValue, _pCalEntry);	
							_nTimeValue := (_nTimeValue+1);
						ELSE
							iOwner.LogMsg.Show1(ADSLOG_MSGTYPE_ERROR, 'RES37', 'Failed to read calendar entry due to insufficient buffer entry limit of "%d entries per calendar"! (See Parameter "nSched_EntryCount")', F_DINT(_nMaxSchedEntryCount), FALSE);
						END_IF		
			
						_pTimeValue:=F_BACnet_NextListElem(_pTimeValue, _pTimeValue^.nEntrySize);
						_pCalEntry := (_pCalEntry+SIZEOF(ST_BA_SchedEntry));
					END_WHILE		
					_nCalEntry := (_nCalEntry+1);
				ELSE
					iOwner.LogMsg.Show1(ADSLOG_MSGTYPE_ERROR, 'RES45', 'Failed to read calendar due to insufficient buffer entry limit of %d! (See Parameter "nSched_CalendarCount")', F_DINT(_nMaxCalCount), FALSE);
				END_IF
			ELSE
				IF (_nExcEntry <= _nMaxExcptCount) THEN
					aException[_nExcEntry].eType := (_pDailySched^.stEvent.eCalEntryChoice+1);
					aException[_nExcEntry].uDate := _pDailySched^.stEvent.uCalEntry;
					aException[_nExcEntry].nEventPriority := _pDailySched^.stEvent.nEventPriority;
					
